			gvl.legCtrl[Mapping23[i]].ForwardKinetics(motorAngles:=OA_FJntRef[i].data , legIndex:=Mapping23[i] , tipPosition=>OA_FPosWrtHip[i].data );
			temp.data[0]:=hip_pos[Mapping23[i],0];temp.data[1]:=hip_pos[Mapping23[i],1];temp.data[2]:=hip_pos[Mapping23[i],2];
			leg_ref_pos[Mapping23[i]]:= VecAdd( MatMulVec(Rb_target1, VecAdd(temp,MatMulVec(Rleg[Mapping23[i]],OA_FPosWrtHip[i]))),body_ref_pos);	
		END_FOR		
	ELSE
		body_ref_pos:=OA_BodyPoseEnd;
		body_ref_ang:=OA_BodyAngEnd;
		leg_ref_pos:=OA_legPosEnterExtract;	
		tr  := (UDINT_TO_LREAL(gait_cycle - EnterOrientAdjustCount) / gvl.sampleRate-2*OA_LiftGroundTime-OA_AdjustTime-OA_AdjustExtractTime )/OA_AdjustExtendTime;
		fbGetPivot(tNow := tr, tTotal := 1.0, pivot => pvt);
		FOR i:=0 TO 1 DO
			FOR j:=0 TO 2 DO
				OA_MJntRef[i].data[j]:=(1-pvt)*OA_MJntExtract[i,j]+pvt*OA_MJntExtend[i,j];
			END_FOR		
			gvl.legCtrl[Mapping14[i]].ForwardKinetics(motorAngles:=OA_MJntRef[i].data , legIndex:=Mapping14[i] , tipPosition=>OA_MPosWrtHip[i].data );
			fbRotMat(yaw := body_ref_ang.data[2], pitch := body_ref_ang.data[1],roll := body_ref_ang.data[0], rm =>  Rb_target1 );
			temp.data[0]:=hip_pos[Mapping14[i],0];temp.data[1]:=hip_pos[Mapping14[i],1];temp.data[2]:=hip_pos[Mapping14[i],2];
			leg_ref_pos[Mapping14[i]]:= VecAdd( MatMulVec(Rb_target1, VecAdd(temp,MatMulVec(Rleg[Mapping14[i]],OA_MPosWrtHip[i]))),body_ref_pos);	

			gvl.legCtrl[Mapping23[i]].ForwardKinetics(motorAngles:=OA_FJntRef[i].data , legIndex:=Mapping23[i] , tipPosition=>OA_FPosWrtHip[i].data );
			temp.data[0]:=hip_pos[Mapping23[i],0];temp.data[1]:=hip_pos[Mapping23[i],1];temp.data[2]:=hip_pos[Mapping23[i],2];
			leg_ref_pos[Mapping23[i]]:= VecAdd( MatMulVec(Rb_target1, VecAdd(temp,MatMulVec(Rleg[Mapping23[i]],OA_FPosWrtHip[i]))),body_ref_pos);		
		END_FOR					
	END_IF
ELSE
	OrientAdjustFinished:=TRUE;
END_IF
END_METHOD

METHOD PUBLIC TrjPlanning_PushReleaseBall : BOOL
VAR_INPUT
END_VAR

VAR
	PushReleaseBall_FJntTarget:ARRAY[0..1,0..2] OF LREAL:=[-90*pi/180,155*pi/180,175*pi/180,
                                                     90*pi/180,155*pi/180,175*pi/180];//prepared position before gripping stone													 
													 
	i,j: INT;
	invalid: LREAL;
	Rb_target1: Mat3;
	temp: vec3;
	flag: INT;
	tr: LREAL;
END_VAR
//push and release method
IF PushReleaseBallFinished=FALSE AND gvl.curlingPushModel=0 THEN
	body_ref_pos:=body_ref_pos_enter;
	body_ref_ang:=body_ref_ang_enter;
	leg_ref_pos:=leg_ref_pos_enter;
	FOR i:=0 TO 1 DO
		IF gait_cycle-EnterPushReleaseBallCount<=PushTime*gvl.sampleRate THEN
			fbHermitInterpolation(t0:=EnterPushReleaseBallCount*delta_t , T:=PushTime , y0:=PushReleaseBall_FPosStartWrtHip[i].data[0] , 
			y1:=PushReleaseBall_FPosStartWrtHip[i].data[0]-PushDistance , v0:=0 , v1:=-PushVelocity , tNow:=(gait_cycle)* delta_t, 
			y=> PushReleaseBall_FPosWrtHip[i].data[0], v=>invalid );
		ELSIF gait_cycle-EnterPushReleaseBallCount<=(PushTime+PRConstVelTime)*gvl.sampleRate THEN
			fbHermitInterpolation(t0:=EnterPushReleaseBallCount*delta_t+PushTime , T:=PRConstVelTime , y0:=PushReleaseBall_FPosStartWrtHip[i].data[0]-PushDistance , 
			y1:=PushReleaseBall_FPosStartWrtHip[i].data[0]-PushDistance-PRConstVelDistance , v0:=-PushVelocity , v1:= -PushVelocity, tNow:=gait_cycle* delta_t, 
			y=> PushReleaseBall_FPosWrtHip[i].data[0], v=>invalid );			
		ELSIF gait_cycle-EnterPushReleaseBallCount<=(PushTime+PRConstVelTime+DecVelTime)*gvl.sampleRate THEN
			fbHermitInterpolation(t0:=EnterPushReleaseBallCount*delta_t+PushTime+PRConstVelTime , T:=DecVelTime , y0:=PushReleaseBall_FPosStartWrtHip[i].data[0]-PushDistance-PRConstVelDistance , 
			y1:=PushReleaseBall_FPosStartWrtHip[i].data[0]-PushDistance-PRConstVelDistance-DecVelDistance , v0:=-PushVelocity , v1:= 0, tNow:=gait_cycle* delta_t, 
			y=> PushReleaseBall_FPosWrtHip[i].data[0], v=>invalid );	
		ELSE
			 PushReleaseBall_FPosWrtHip[i].data[0]:=PushReleaseBall_FPosStartWrtHip[i].data[0]-PushDistance-PRConstVelDistance-DecVelDistance;	
			 PushReleaseBallFinished:=TRUE;	
			 EnterPushFinishCount:=gait_cycle;
			 
		END_IF
		PushReleaseBall_FPosWrtHip[i].data[1]:=PushReleaseBall_FPosStartWrtHip[i].data[1];
		PushReleaseBall_FPosWrtHip[i].data[2]:=PushReleaseBall_FPosStartWrtHip[i].data[2];
		
		fbRotMat(yaw := body_ref_ang_enter.data[2], pitch := body_ref_ang_enter.data[1],roll := body_ref_ang_enter.data[0], rm =>  Rb_target1 );
		temp.data[0]:=hip_pos[Mapping23[i],0];temp.data[1]:=hip_pos[Mapping23[i],1];temp.data[2]:=hip_pos[Mapping23[i],2];
		leg_ref_pos[Mapping23[i]]:= VecAdd( MatMulVec(Rb_target1, VecAdd(temp,MatMulVec(Rleg[Mapping23[i]],PushReleaseBall_FPosWrtHip[i]))),body_ref_pos);
	END_FOR
END_IF



//only release method
IF PushReleaseBallFinished=FALSE AND gvl.curlingPushModel=1 THEN
	IF gait_cycle - EnterPushReleaseBallCount<=ReleaseTime*gvl.sampleRate THEN
		body_ref_pos:=body_ref_pos_enter;
		body_ref_ang:=body_ref_ang_enter;
		leg_ref_pos:=leg_ref_pos_enter;
	
		tr  := UDINT_TO_LREAL(gait_cycle - EnterPushReleaseBallCount) / gvl.sampleRate / ReleaseTime;
		fbGetPivot(tNow := tr, tTotal := 1.0, pivot => pvt);
		FOR i:=0 TO 1 DO
			FOR j:=0 TO 2 DO
				PushReleaseBall_FJntRef[i].data[j]:=(1-pvt)*PushReleaseBall_FJntStart[i].data[j]+pvt*(PushReleaseBall_FJntTarget[i,j]);
			END_FOR
			gvl.legCtrl[Mapping23[i]].ForwardKinetics(motorAngles:=PushReleaseBall_FJntRef[i].data , legIndex:=Mapping23[i] , tipPosition=>PushReleaseBall_FPosWrtHip[i].data );
			fbRotMat(yaw := body_ref_ang_enter.data[2], pitch := body_ref_ang_enter.data[1],roll := body_ref_ang_enter.data[0], rm =>  Rb_target1 );
			temp.data[0]:=hip_pos[Mapping23[i],0];temp.data[1]:=hip_pos[Mapping23[i],1];temp.data[2]:=hip_pos[Mapping23[i],2];
			leg_ref_pos[Mapping23[i]]:= VecAdd( MatMulVec(Rb_target1, VecAdd(temp,MatMulVec(Rleg[Mapping23[i]],PushReleaseBall_FPosWrtHip[i]))),body_ref_pos);
		END_FOR
	ELSE	
		PushReleaseBallFinished:=TRUE;
		EnterPushFinishCount:=gait_cycle;
	END_IF	
END_IF

IF PushReleaseBallFinished=TRUE AND SpeedDownFinished=FALSE AND gait_cycle-EnterPushFinishCount>=LREAL_TO_UDINT(PushFinishDurationTime)*gvl.sampleRate  THEN
	RequireSpeedDown:=TRUE;
END_IF
END_METHOD

METHOD PUBLIC TrjPlanning_Recovery : BOOL
VAR_INPUT
END_VAR
VAR
	legExtractRefPosCurling: ARRAY[0..5, 0..2] OF LREAL:=[-0.35,-0.3+0.02,0,
														  0.1,-0.3+0.02,-0.1246,
														  -0.3+0.05,-0.3+0.02,-0.1246,
														  -0.3+0.05,-0.3+0.02,0.1246,
														  0.1,-0.3+0.02,0.1246,
														  -0.35,-0.3+0.02,0];//-0.15 for front leg
	jntExtractRefPosCurling: ARRAY[0..5, 0..2] OF LREAL:=[0,163.1808*pi/180,297.208*pi/180,
											  			  0,322.9120*pi/180,(205.1705-322.9120)*pi/180,
											              0,183.8227*pi/180,(269.8634-183.8227)*pi/180,
											              0,183.8227*pi/180,(269.8634-183.8227)*pi/180,
											              0,322.9120*pi/180,(205.1705-322.9120)*pi/180,
											              0,163.1808*pi/180,297.208*pi/180];
	legExtendRefPosCurling: ARRAY[0..5, 0..2] OF LREAL:=[-0.35,-0.4-0.07,0,
														  0.1,-0.4-0.07,-0.1246,
														  -0.3+0.05,-0.4-0.07,-0.1246,
														  -0.3+0.05,-0.4-0.07,0.1246,
														  0.1,-0.4-0.07,0.1246,
														  -0.35,-0.4-0.07,0];	//-0.15 for front leg													 
	jntExtendRefPosCurling: ARRAY[0..5, 0..2] OF LREAL:=[0,181.9845*pi/180,299.9603*pi/180,
											 			 0,302.7132*pi/180,(230.9946-302.7132)*pi/180,	
											             0,222.0252*pi/180,(254.0072-222.0252)*pi/180,
											             0,222.0252*pi/180,(254.0072-222.0252)*pi/180,
									                     0,302.7132*pi/180,(230.9946-302.7132)*pi/180,
											             0,181.9845*pi/180,299.9603*pi/180]	;

	(*legExtractRefPosCurling:    ARRAY[0..5, 0..2] OF LREAL:=[-0.35,-0.3+0.08,0,
														  0.1,-0.3209+0.08,-0.1246,
														  -0.3,-0.3209+0.08,-0.1246,
														  -0.3,-0.3209+0.08,0.1246,
														  0.1,-0.3209+0.08,0.1246,
														  -0.35,-0.3+0.08,0];															  
	jntExtractRefPosCurling: ARRAY[0..5, 0..2] OF LREAL:= [0,150.7997*pi/180,291.8958*pi/180,
											  			0,327.8142*pi/180,(196.8366-327.8142)*pi/180,
											  			0,172.5134*pi/180,(269.4767-172.5134)*pi/180,
											  			0,172.5134*pi/180,(269.4767-172.5134)*pi/180,
											  			0,327.8142*pi/180,(196.8366-327.8142)*pi/180,
											  			0,150.7997*pi/180,291.8958*pi/180];	
	legExtendRefPosCurling: ARRAY[0..5, 0..2] OF LREAL    :=[-0.35,-0.3209,0,
														  0.1,-0.3209,-0.1246,
														  -0.3,-0.3209,-0.1246,
														  -0.3,-0.3209,0.1246,
														  0.1,-0.3209,0.1246,
														  -0.35,-0.3209,0];														  													  
	jntExtendRefPosCurling: ARRAY[0..5, 0..2] OF LREAL:=	[0,163.1808*pi/180,297.208*pi/180,
											 				0,320.9331*pi/180,(208.0880-320.9331)*pi/180,	
											 				0,187.8384*pi/180,(269.4264-187.8384)*pi/180,
															0,187.8384*pi/180,(269.4264-187.8384)*pi/180,
									         				0,320.9331*pi/180,(208.0880-320.9331)*pi/180,
											 				0,163.1808*pi/180,297.208*pi/180];*)
													  
	i: INT;
	j: INT;
	tempLeg:ARRAY [0..2] OF LREAL;
	tempJnt:ARRAY [0..2] OF LREAL;
	tempRef:ARRAY [0..2] OF LREAL;
	tTotal: LREAL;
	tNow: LREAL;
	jntPosBegin : ARRAY[0..5, 0..2] OF LREAL;
	jntPosEnd   : ARRAY[0..5, 0..2] OF LREAL;
	Rb_target1: Mat3;
	temp: vec3;
	tipForceDesireGroupA:ARRAY[0..5,0..2] OF LREAL:=[0,-100,0,
													 0,0,0,
													 0,0,0,
													 0,0,0,
													 0,0,0,
													 0,0,0];
	tipForceDesireGroupB:ARRAY[0..5,0..2] OF LREAL:=[0,0,0,
													 0,0,0,
													 0,0,0,
													 0,0,0,
													 0,0,0,
													 0,-120,0];
	tr: LREAL;
END_VAR
IF (gait_cycle-EnterRecoveryCount)=1 THEN
	FOR i:=0 TO 5 DO
		tempLeg[0]:=legExtractRefPosCurling[i,0];tempLeg[1]:=legExtractRefPosCurling[i,1];tempLeg[2]:=legExtractRefPosCurling[i,2];
		tempRef[0]:=jntExtractRefPosCurling[i,0];tempRef[1]:=jntExtractRefPosCurling[i,1];tempRef[2]:=jntExtractRefPosCurling[i,2];
		GVL.legCtrl[i].InverseKinetics(tipPosition:=tempLeg , refPosLast:=tempRef , legIndex:=i , motorAngles=>tempJnt , isSingular=> );
		jntAngRetract[i,0]:=tempJnt[0];jntAngRetract[i,1]:=tempJnt[1];jntAngRetract[i,2]:=tempJnt[2];
		
		tempLeg[0]:=legExtendRefPosCurling[i,0];tempLeg[1]:=legExtendRefPosCurling[i,1];tempLeg[2]:=legExtendRefPosCurling[i,2];
		tempRef[0]:=jntExtendRefPosCurling[i,0];tempRef[1]:=jntExtendRefPosCurling[i,1];tempRef[2]:=jntExtendRefPosCurling[i,2];
		GVL.legCtrl[i].InverseKinetics(tipPosition:=tempLeg , refPosLast:=tempRef , legIndex:=i , motorAngles=>tempJnt , isSingular=> );
		jntAngExtend[i,0]:=tempJnt[0];jntAngExtend[i,1]:=tempJnt[1];jntAngExtend[i,2]:=tempJnt[2];			
		
	END_FOR
	tipForceDesire:=tipForceDesireZeros;

END_IF

IF RecoveryFinished=FALSE THEN
	body_ref_pos:=body_ref_pos_enter;
	body_ref_ang:=body_ref_ang_enter;
	leg_ref_pos:=leg_ref_pos_enter;
	
	IF (gait_cycle-EnterRecoveryCount)<=(tRetract + tWait + tExtend) * gvl.sampleRate THEN //leg 0-2-4 recovery
		
		//force compensator****************************
		IF (gait_cycle-EnterRecoveryCount)<=fceLoadTime*gvl.sampleRate THEN
			tr  := UDINT_TO_LREAL(gait_cycle-EnterRecoveryCount) / gvl.sampleRate /fceLoadTime;
			fbGetPivot(tNow := tr, tTotal := 1.0, pivot => pvt);
			FOR i:=0 TO 5 DO
				FOR j:=0 TO 2 DO
					tipForceDesire[i,j]:=(1-pvt)*tipForceDesireZeros[i,j]+pvt*tipForceDesireGroupB[i,j];//group B add load
				END_FOR
			END_FOR
		ELSIF  (gait_cycle-EnterRecoveryCount)>LREAL_TO_UDINT((tRetract + tWait + tExtend-fceLoadTime)*gvl.sampleRate) AND  (gait_cycle-EnterRecoveryCount)<=LREAL_TO_UDINT((tRetract + tWait + tExtend) * gvl.sampleRate) THEN
			tr  := (UDINT_TO_LREAL (gait_cycle-EnterRecoveryCount) / gvl.sampleRate-(tRetract + tWait + tExtend-fceLoadTime) )/fceLoadTime;
			fbGetPivot(tNow := tr, tTotal := 1.0, pivot => pvt);
			FOR i:=0 TO 5 BY 2DO
				FOR j:=0 TO 2 DO
					//tipForceDesire[i,j]:=(1-pvt)*tipForceDesireZeros[i,j]+pvt*tipForceDesireGroupA[i,j];//group A add load
					tipForceDesire[i+1,j]:=(1-pvt)*tipForceDesireGroupB[i+1,j]+pvt*tipForceDesireZeros[i+1,j];//group B reduce load
				END_FOR
			END_FOR
		ELSE
		tipForceDesire:=tipForceDesireGroupB;
		END_IF
		//***********************************************
	
		IF gait_cycle-EnterRecoveryCount < tRetract * gvl.sampleRate THEN
			tTotal := tRetract;
			tNow   := UDINT_TO_LREAL(gait_cycle-EnterRecoveryCount) * 1.0 / DINT_TO_LREAL(gvl.sampleRate);
			jntPosBegin := RcJointPosStart;
			FOR i:=0 TO 5 BY 2 DO
				FOR j:=0 TO 2 DO
					jntPosEnd[i,j]:=jntAngRetract[i,j];
					jntPosEnd[i+1,j]:=RcJointPosStart[i+1,j];
				END_FOR
			END_FOR
		ELSIF gait_cycle-EnterRecoveryCount  < (tRetract + tWait) * gvl.sampleRate THEN
			tTotal := tWait;
			tNow   := UDINT_TO_LREAL(gait_cycle-EnterRecoveryCount) * 1.0 / DINT_TO_LREAL(gvl.sampleRate) - tRetract;
			FOR i:=0 TO 5 BY 2 DO
				FOR j:=0 TO 2 DO
					jntPosBegin[i,j]:=jntAngRetract[i,j];
					jntPosBegin[i+1,j]:=RcJointPosStart[i+1,j];
					jntPosEnd[i,j]:=jntAngRetract[i,j];
					jntPosEnd[i+1,j]:=RcJointPosStart[i+1,j];
				END_FOR
			END_FOR
		ELSE 
			tTotal := tExtend;
			tNow   := UDINT_TO_LREAL(gait_cycle-EnterRecoveryCount) * 1.0 / DINT_TO_LREAL(gvl.sampleRate) - tRetract - tWait;
			FOR i:=0 TO 5 BY 2 DO
				FOR j:=0 TO 2 DO
					jntPosBegin[i,j]:=jntAngRetract[i,j];
					jntPosBegin[i+1,j]:=RcJointPosStart[i+1,j];
					jntPosEnd[i,j]:=jntAngExtend[i,j];
					jntPosEnd[i+1,j]:=RcJointPosStart[i+1,j];
				END_FOR
			END_FOR	
		END_IF	
	ELSIF (gait_cycle-EnterRecoveryCount)<=2*(tRetract + tWait + tExtend) * gvl.sampleRate  THEN //leg 1-3-5 recovery

		//force compensator*******************
		IF (gait_cycle-EnterRecoveryCount)>LREAL_TO_UDINT((tRetract + tWait + tExtend)*gvl.sampleRate) AND (gait_cycle-EnterRecoveryCount)<=LREAL_TO_UDINT((tRetract + tWait + tExtend+fceLoadTime)* gvl.sampleRate) THEN
			tr  := (UDINT_TO_LREAL(gait_cycle-EnterRecoveryCount) / gvl.sampleRate-(tRetract + tWait + tExtend) )/fceLoadTime;
			fbGetPivot(tNow := tr, tTotal := 1.0, pivot => pvt);
			FOR i:=0 TO 5 BY 2 DO
				FOR j:=0 TO 2 DO
					tipForceDesire[i,j]:=(1-pvt)*tipForceDesireZeros[i,j]+pvt*tipForceDesireGroupA[i,j];//group A add load
					tipForceDesire[i+1,j]:=tipForceDesireZeros[i+1,j];//group B zeros load
				END_FOR
			END_FOR		
		ELSIF (gait_cycle-EnterRecoveryCount)>LREAL_TO_UDINT((2*(tRetract + tWait + tExtend)-fceLoadTime)*gvl.sampleRate) AND (gait_cycle-EnterRecoveryCount)<=LREAL_TO_UDINT(2*(tRetract + tWait + tExtend) * gvl.sampleRate) THEN
			tr  := (UDINT_TO_LREAL(gait_cycle-EnterRecoveryCount) / gvl.sampleRate-(2*(tRetract + tWait + tExtend)-fceLoadTime) )/fceLoadTime;
			fbGetPivot(tNow := tr, tTotal := 1.0, pivot => pvt);
			FOR i:=0 TO 5 BY 2DO
				FOR j:=0 TO 2 DO
					tipForceDesire[i,j]:=(1-pvt)*tipForceDesireGroupA[i,j]+pvt*tipForceDesireZeros[i,j];//group A reduce load
					tipForceDesire[i+1,j]:=tipForceDesireZeros[i+1,j];//group B zeros load
				END_FOR
			END_FOR	
		ELSE	
			tipForceDesire:=tipForceDesireGroupA;
		END_IF	
		//******************************************	

		
		IF gait_cycle-EnterRecoveryCount<=(2*tRetract + tWait + tExtend) * gvl.sampleRate THEN
			tTotal := tRetract;
			tNow   := UDINT_TO_LREAL(gait_cycle-EnterRecoveryCount) * 1.0 / DINT_TO_LREAL(gvl.sampleRate)-(tRetract + tWait + tExtend);
			FOR i:=0 TO 5 BY 2 DO
				FOR j:=0 TO 2 DO
					jntPosBegin[i,j]:=jntAngExtend[i,j];
					jntPosBegin[i+1,j]:=RcJointPosStart[i+1,j];
					jntPosEnd[i,j]:=jntAngExtend[i,j];
					jntPosEnd[i+1,j]:=jntAngRetract[i+1,j];
				END_FOR
			END_FOR			
		ELSIF gait_cycle-EnterRecoveryCount<=(2*tRetract + 2*tWait + tExtend) * gvl.sampleRate THEN
			tTotal := tWait;
			tNow   := UDINT_TO_LREAL(gait_cycle-EnterRecoveryCount) * 1.0 / DINT_TO_LREAL(gvl.sampleRate) - (2*tRetract + tWait + tExtend);
			FOR i:=0 TO 5 BY 2 DO
				FOR j:=0 TO 2 DO
					jntPosBegin[i,j]:=jntAngExtend[i,j];
					jntPosBegin[i+1,j]:=jntAngRetract[i+1,j];
					jntPosEnd[i,j]:=jntAngExtend[i,j];
					jntPosEnd[i+1,j]:=jntAngRetract[i+1,j];
				END_FOR
			END_FOR			
		ELSE
			tTotal := tExtend;
			tNow   := UDINT_TO_LREAL(gait_cycle-EnterRecoveryCount) * 1.0 / DINT_TO_LREAL(gvl.sampleRate) - (2*tRetract + 2*tWait + tExtend);
			FOR i:=0 TO 5 BY 2 DO
				FOR j:=0 TO 2 DO
					jntPosBegin[i,j]:=jntAngExtend[i,j];
					jntPosBegin[i+1,j]:=jntAngRetract[i+1,j];
					jntPosEnd[i,j]:=jntAngExtend[i,j];
					jntPosEnd[i+1,j]:=jntAngExtend[i+1,j];
				END_FOR
			END_FOR			
		END_IF
	ELSE
		tTotal := 100;
		tNow   := UDINT_TO_LREAL(gait_cycle-EnterRecoveryCount) * 1.0 / DINT_TO_LREAL(gvl.sampleRate) - 2*tRetract - 2*tWait - 2*tExtend;
		jntPosBegin :=jntAngExtend;
		jntPosEnd :=jntAngExtend;
		RecoveryFinished:=TRUE;
		tipForceDesire:=tipForceDesireZeros;
		RequireReduceHeightB:=TRUE;
	END_IF
	getPivot(tNow := tNow, tTotal := tTotal, pivot => pivot, pivotDot => pivotDot);
	FOR i := 0 TO 5 DO
		FOR j := 0 TO 2 DO
			RcJointPosRef[i, j] := (1.0 - pivot) * jntPosBegin[i, j] + pivot * jntPosEnd[i, j];
		END_FOR
		tempJnt[0]:=RcJointPosRef[i,0];tempJnt[1]:=RcJointPosRef[i,1];tempJnt[2]:=RcJointPosRef[i,2];
		gvl.legCtrl[i].ForwardKinetics(motorAngles:=tempJnt , legIndex:=i , tipPosition=>Rc_PosWrtHip[i].data );
		fbRotMat(yaw := body_ref_ang_enter.data[2], pitch := body_ref_ang_enter.data[1],roll := body_ref_ang_enter.data[0], rm =>  Rb_target1 );
		temp.data[0]:=hip_pos[i,0];temp.data[1]:=hip_pos[i,1];temp.data[2]:=hip_pos[i,2];
		leg_ref_pos[i]:= VecAdd( MatMulVec(Rb_target1, VecAdd(temp,MatMulVec(Rleg[i],Rc_PosWrtHip[i]))),body_ref_pos);		
	END_FOR

END_IF
END_METHOD

METHOD PUBLIC TrjPlanning_ReduceHeight : BOOL
VAR_INPUT
	
END_VAR
VAR
	
	tr: LREAL;
	i: INT;
	Rb_target1: Mat3;
	temp: vec3;
END_VAR
IF ReduceHeightFinished=FALSE AND (gait_cycle-EnterReduceHeightCount)<=ReduceHeightTime*gvl.sampleRate THEN
	body_ref_ang:=body_ref_ang_enter;
	leg_ref_pos:=leg_ref_pos_enter;
	tr  := UDINT_TO_LREAL(gait_cycle - EnterReduceHeightCount) / gvl.sampleRate / ReduceHeightTime;
	fbGetPivot(tNow := tr, tTotal := 1.0, pivot => pvt);
	FOR i:=0 TO 2 DO
		body_ref_pos.data[i]:=(1-pvt)*body_ref_pos_enter.data[i]+pvt*body_target_pos.data[i];
	END_FOR
	FOR i:=0 TO 1 DO
		gvl.legCtrl[Mapping23[i]].ForwardKinetics(motorAngles:=ReduceHeight_FJntRef[i].data , legIndex:=Mapping23[i] , tipPosition=>ReduceHeight_FPosWrtHip[i].data );
		fbRotMat(yaw := body_ref_ang_enter.data[2], pitch := body_ref_ang_enter.data[1],roll := body_ref_ang_enter.data[0], rm =>  Rb_target1 );
		temp.data[0]:=hip_pos[Mapping23[i],0];temp.data[1]:=hip_pos[Mapping23[i],1];temp.data[2]:=hip_pos[Mapping23[i],2];
		leg_ref_pos[Mapping23[i]]:= VecAdd( MatMulVec(Rb_target1, VecAdd(temp,MatMulVec(Rleg[Mapping23[i]],ReduceHeight_FPosWrtHip[i]))),body_ref_pos);
	END_FOR
ELSE
	ReduceHeightFinished:=TRUE;
END_IF
END_METHOD

METHOD PUBLIC TrjPlanning_ReduceHeightB : BOOL
VAR_INPUT
END_VAR
VAR
	tr: LREAL;
	i: INT;
	Rb_target1: Mat3;
	temp: vec3;
END_VAR
IF ReduceHeightBFinished=FALSE AND (gait_cycle-EnterReduceHeightBCount)<=RHB_time*gvl.sampleRate THEN
	body_ref_ang:=body_ref_ang_enter;
	leg_ref_pos:=leg_ref_pos_enter;
	tr  := UDINT_TO_LREAL(gait_cycle - EnterReduceHeightBCount) / gvl.sampleRate / RHB_time;
	fbGetPivot(tNow := tr, tTotal := 1.0, pivot => pvt);
	FOR i:=0 TO 2 DO
		body_ref_pos.data[i]:=(1-pvt)*body_ref_pos_enter.data[i]+pvt*RHB_body_target_pos.data[i];
	END_FOR
ELSE
	ReduceHeightBFinished:=TRUE;
END_IF
END_METHOD

METHOD PUBLIC TrjPlanning_SearchPedal : BOOL
VAR_INPUT
END_VAR
VAR
	tr: LREAL;
	i: INT;
	j: INT;
	Rb_target1: Mat3;
	temp: vec3;
	
	tipForceDesireLegA:	 ARRAY[0..5,0..2] OF LREAL:=[0,-100,0,
													 0,0,0,
													 0,0,0,
													 0,0,0,
													 0,0,0,
													 0,0,0];
	tipForceDesireLegF:	 ARRAY[0..5,0..2] OF LREAL:=[0,0,0,
													 0,0,0,
													 0,0,0,
													 0,0,0,
													 0,0,0,
													 0,-120,0];				
END_VAR
IF SearchPedalFinished=FALSE THEN
	IF SP_RBLegSearching=TRUE THEN
		SP_LBLegSearching:=FALSE;
		body_ref_pos:=body_ref_pos_enter;
		body_ref_ang:=body_ref_ang_enter;
		leg_ref_pos:=leg_ref_pos_enter;	
		IF (gait_cycle-SP_EnterSubSearchCount[0])<=SP_LiftLegTime*gvl.sampleRate THEN
			tr  := UDINT_TO_LREAL(gait_cycle - SP_EnterSubSearchCount[0]) / gvl.sampleRate / SP_LiftLegTime;
			fbGetPivot(tNow := tr, tTotal := 1.0, pivot => pvt);	
			SP_BPosRefWrtHip[0].data[0]:=SP_BPosStartWrtHip[0].data[0];
			SP_BPosRefWrtHip[0].data[1]:=(1-pvt)*SP_BPosStartWrtHip[0].data[1]+pvt*(SP_BPosStartWrtHip[0].data[1]+SP_LiftDistance);
			SP_BPosRefWrtHip[0].data[2]:=SP_BPosStartWrtHip[0].data[2];
			fbRotMat(yaw := body_ref_ang_enter.data[2], pitch := body_ref_ang_enter.data[1],roll := body_ref_ang_enter.data[0], rm =>  Rb_target1 );
			temp.data[0]:=hip_pos[0,0];temp.data[1]:=hip_pos[0,1];temp.data[2]:=hip_pos[0,2];
			leg_ref_pos[0]:= VecAdd( MatMulVec(Rb_target1, VecAdd(temp,MatMulVec(Rleg[0],SP_BPosRefWrtHip[0]))),body_ref_pos);	
			
			//force compensator
			tipForceTarget:=tipForceDesireLegF;
			IF (gait_cycle-SP_EnterSubSearchCount[0])<=LREAL_TO_UDINT(fceLoadTime*gvl.sampleRate) THEN
				tr  := (UDINT_TO_LREAL(gait_cycle-SP_EnterSubSearchCount[0]) / gvl.sampleRate)/ fceLoadTime;
				fbGetPivot(tNow := tr, tTotal := 1.0, pivot => pvt);
				FOR i:=0 TO 5 DO
					FOR j:=0 TO 2 DO
						tipForceDesire[i,j]:=(1-pvt)*tipForceDesireZeros[i,j]+pvt*tipForceTarget[i,j];
					END_FOR
				END_FOR
			END_IF
			
		ELSIF (gait_cycle-SP_EnterSubSearchCount[0])<=(SP_LiftLegTime+SP_SearchTime)*gvl.sampleRate AND  SP_BLegSearchFinished[0]=FALSE THEN
			tr  := (UDINT_TO_LREAL(gait_cycle - SP_EnterSubSearchCount[0]) / gvl.sampleRate -SP_LiftLegTime)/ SP_SearchTime;
			fbGetPivot(tNow := tr, tTotal := 1.0, pivot => pvt);	
			SP_BPosRefWrtHip[0].data[0]:=(1-pvt)*SP_BPosStartWrtHip[0].data[0]+pvt*(SP_BPosStartWrtHip[0].data[0]-SP_SearchDistance);		
			SP_BPosRefWrtHip[0].data[1]:=SP_BPosStartWrtHip[0].data[1]+SP_LiftDistance;
			SP_BPosRefWrtHip[0].data[2]:=SP_BPosStartWrtHip[0].data[2];
			IF isPedal(0)=TRUE AND  SP_BLegSearchFinished[0]=FALSE THEN
				SP_BLegSearchFinished[0]:=TRUE;
				SP_EnterSubSearchDecreaseCount[0]:=gait_cycle;
				FOR j:=0 TO 2 DO
					SP_BPosLockWrtHip[0].data[j]:=SP_BPosRefWrtHip[0].data[j];
				END_FOR			
			END_IF
			IF (gait_cycle-SP_EnterSubSearchCount[0])=LREAL_TO_UDINT((SP_LiftLegTime+SP_SearchTime)*gvl.sampleRate) AND SP_BLegSearchFinished[0]=FALSE THEN
				SP_BLegSearchFinished[0]:=TRUE;
				SP_EnterSubSearchDecreaseCount[0]:=gait_cycle;
				FOR j:=0 TO 2 DO
					SP_BPosLockWrtHip[0].data[j]:=SP_BPosRefWrtHip[0].data[j];
				END_FOR	
			END_IF

			fbRotMat(yaw := body_ref_ang_enter.data[2], pitch := body_ref_ang_enter.data[1],roll := body_ref_ang_enter.data[0], rm =>  Rb_target1 );
			temp.data[0]:=hip_pos[0,0];temp.data[1]:=hip_pos[0,1];temp.data[2]:=hip_pos[0,2];
			leg_ref_pos[0]:= VecAdd( MatMulVec(Rb_target1, VecAdd(temp,MatMulVec(Rleg[0],SP_BPosRefWrtHip[0]))),body_ref_pos);	
			
		ELSIF  SP_BLegSearchFinished[0]=TRUE AND (gait_cycle-SP_EnterSubSearchDecreaseCount[0])<=SP_LiftLegTime*gvl.sampleRate THEN
			tr  := UDINT_TO_LREAL(gait_cycle - SP_EnterSubSearchDecreaseCount[0]) / gvl.sampleRate / SP_LiftLegTime;
			fbGetPivot(tNow := tr, tTotal := 1.0, pivot => pvt);
			SP_BPosRefWrtHip[0].data[0]:=SP_BPosLockWrtHip[0].data[0];	
			SP_BPosRefWrtHip[0].data[1]:=(1-pvt)*SP_BPosLockWrtHip[0].data[1]+pvt*(SP_BPosLockWrtHip[0].data[1]-SP_LiftDistance);
			SP_BPosRefWrtHip[0].data[2]:=SP_BPosLockWrtHip[0].data[2];	
			
			fbRotMat(yaw := body_ref_ang_enter.data[2], pitch := body_ref_ang_enter.data[1],roll := body_ref_ang_enter.data[0], rm =>  Rb_target1 );
			temp.data[0]:=hip_pos[0,0];temp.data[1]:=hip_pos[0,1];temp.data[2]:=hip_pos[0,2];
			leg_ref_pos[0]:= VecAdd( MatMulVec(Rb_target1, VecAdd(temp,MatMulVec(Rleg[0],SP_BPosRefWrtHip[0]))),body_ref_pos);	
			IF (gait_cycle-SP_EnterSubSearchDecreaseCount[0])=LREAL_TO_UDINT( SP_LiftLegTime*gvl.sampleRate) THEN
				body_ref_pos_enter:=body_ref_pos;
				body_ref_ang_enter:=body_ref_ang;
				leg_ref_pos_enter:=leg_ref_pos;	
			END_IF	
			
			//force compensator
			tipForceTarget:=tipForceDesireLegF;
			IF (gait_cycle-SP_EnterSubSearchDecreaseCount[0])>LREAL_TO_UDINT((SP_LiftLegTime-fceLoadTime)*gvl.sampleRate)THEN
				tr  := (UDINT_TO_LREAL(gait_cycle-SP_EnterSubSearchDecreaseCount[0]) / gvl.sampleRate-(SP_LiftLegTime-fceLoadTime) )/ fceLoadTime;
				fbGetPivot(tNow := tr, tTotal := 1.0, pivot => pvt);
				FOR i:=0 TO 5 DO
					FOR j:=0 TO 2 DO
						tipForceDesire[i,j]:=(1-pvt)*tipForceTarget[i,j]+pvt*tipForceDesireZeros[i,j];
					END_FOR
				END_FOR
			END_IF
	
		ELSE
			SP_RBLegSearching:=FALSE;
			SP_LBLegSearching:=TRUE;
			SP_EnterSubSearchCount[1]:=gait_cycle;			
		END_IF
	END_IF
	
	IF SP_LBLegSearching=TRUE THEN
		SP_RBLegSearching:=FALSE;
		body_ref_pos:=body_ref_pos_enter;
		body_ref_ang:=body_ref_ang_enter;
		leg_ref_pos:=leg_ref_pos_enter;	
		IF (gait_cycle-SP_EnterSubSearchCount[1])<=SP_LiftLegTime*gvl.sampleRate THEN
			tr  := UDINT_TO_LREAL(gait_cycle - SP_EnterSubSearchCount[1]) / gvl.sampleRate / SP_LiftLegTime;
			fbGetPivot(tNow := tr, tTotal := 1.0, pivot => pvt);	
			SP_BPosRefWrtHip[1].data[0]:=SP_BPosStartWrtHip[1].data[0];
			SP_BPosRefWrtHip[1].data[1]:=(1-pvt)*SP_BPosStartWrtHip[1].data[1]+pvt*(SP_BPosStartWrtHip[1].data[1]+SP_LiftDistance);
			SP_BPosRefWrtHip[1].data[2]:=SP_BPosStartWrtHip[1].data[2];
			fbRotMat(yaw := body_ref_ang_enter.data[2], pitch := body_ref_ang_enter.data[1],roll := body_ref_ang_enter.data[0], rm =>  Rb_target1 );
			temp.data[0]:=hip_pos[5,0];temp.data[1]:=hip_pos[5,1];temp.data[2]:=hip_pos[5,2];
			leg_ref_pos[5]:= VecAdd( MatMulVec(Rb_target1, VecAdd(temp,MatMulVec(Rleg[5],SP_BPosRefWrtHip[1]))),body_ref_pos);	
			
			//force compensator
			tipForceTarget:=tipForceDesireLegA;
			IF (gait_cycle-SP_EnterSubSearchCount[1])<=LREAL_TO_UDINT(fceLoadTime*gvl.sampleRate) THEN
				tr  := (UDINT_TO_LREAL(gait_cycle-SP_EnterSubSearchCount[1]) / gvl.sampleRate)/ fceLoadTime;
				fbGetPivot(tNow := tr, tTotal := 1.0, pivot => pvt);
				FOR i:=0 TO 5 DO
					FOR j:=0 TO 2 DO
						tipForceDesire[i,j]:=(1-pvt)*tipForceDesireZeros[i,j]+pvt*tipForceTarget[i,j];
					END_FOR
				END_FOR
			END_IF
			
		ELSIF (gait_cycle-SP_EnterSubSearchCount[1])<=(SP_LiftLegTime+SP_SearchTime)*gvl.sampleRate AND  SP_BLegSearchFinished[1]=FALSE THEN
			tr  := (UDINT_TO_LREAL(gait_cycle - SP_EnterSubSearchCount[1]) / gvl.sampleRate -SP_LiftLegTime)/ SP_SearchTime;
			fbGetPivot(tNow := tr, tTotal := 1.0, pivot => pvt);	
			SP_BPosRefWrtHip[1].data[0]:=(1-pvt)*SP_BPosStartWrtHip[1].data[0]+pvt*(SP_BPosStartWrtHip[1].data[0]-SP_SearchDistance);		
			SP_BPosRefWrtHip[1].data[1]:=SP_BPosStartWrtHip[1].data[1]+SP_LiftDistance;
			SP_BPosRefWrtHip[1].data[2]:=SP_BPosStartWrtHip[1].data[2];
			IF isPedal(5)=TRUE AND  SP_BLegSearchFinished[1]=FALSE THEN
				SP_BLegSearchFinished[1]:=TRUE;
				SP_EnterSubSearchDecreaseCount[1]:=gait_cycle;
				FOR j:=0 TO 2 DO
					SP_BPosLockWrtHip[1].data[j]:=SP_BPosRefWrtHip[1].data[j];
				END_FOR			
			END_IF
			IF (gait_cycle-SP_EnterSubSearchCount[1])=LREAL_TO_UDINT((SP_LiftLegTime+SP_SearchTime)*gvl.sampleRate) AND SP_BLegSearchFinished[1]=FALSE THEN
				SP_BLegSearchFinished[1]:=TRUE;
				SP_EnterSubSearchDecreaseCount[1]:=gait_cycle;
				FOR j:=0 TO 2 DO
					SP_BPosLockWrtHip[1].data[j]:=SP_BPosRefWrtHip[1].data[j];
				END_FOR	
			END_IF

			fbRotMat(yaw := body_ref_ang_enter.data[2], pitch := body_ref_ang_enter.data[1],roll := body_ref_ang_enter.data[0], rm =>  Rb_target1 );
			temp.data[0]:=hip_pos[5,0];temp.data[1]:=hip_pos[5,1];temp.data[2]:=hip_pos[5,2];
			leg_ref_pos[5]:= VecAdd( MatMulVec(Rb_target1, VecAdd(temp,MatMulVec(Rleg[5],SP_BPosRefWrtHip[1]))),body_ref_pos);	
			
		ELSIF  SP_BLegSearchFinished[1]=TRUE AND (gait_cycle-SP_EnterSubSearchDecreaseCount[1])<=SP_LiftLegTime*gvl.sampleRate THEN
			tr  := UDINT_TO_LREAL(gait_cycle - SP_EnterSubSearchDecreaseCount[1]) / gvl.sampleRate / SP_LiftLegTime;
			fbGetPivot(tNow := tr, tTotal := 1.0, pivot => pvt);
			SP_BPosRefWrtHip[1].data[0]:=SP_BPosLockWrtHip[1].data[0];	
			SP_BPosRefWrtHip[1].data[1]:=(1-pvt)*SP_BPosLockWrtHip[1].data[1]+pvt*(SP_BPosLockWrtHip[1].data[1]-SP_LiftDistance);
			SP_BPosRefWrtHip[1].data[2]:=SP_BPosLockWrtHip[1].data[2];	
			
			fbRotMat(yaw := body_ref_ang_enter.data[2], pitch := body_ref_ang_enter.data[1],roll := body_ref_ang_enter.data[0], rm =>  Rb_target1 );
			temp.data[0]:=hip_pos[5,0];temp.data[1]:=hip_pos[5,1];temp.data[2]:=hip_pos[5,2];
			leg_ref_pos[5]:= VecAdd( MatMulVec(Rb_target1, VecAdd(temp,MatMulVec(Rleg[5],SP_BPosRefWrtHip[1]))),body_ref_pos);	
			IF (gait_cycle-SP_EnterSubSearchDecreaseCount[1])=LREAL_TO_UDINT( SP_LiftLegTime*gvl.sampleRate) THEN
				body_ref_pos_enter:=body_ref_pos;
				body_ref_ang_enter:=body_ref_ang;
				leg_ref_pos_enter:=leg_ref_pos;	
			END_IF	
			
			//force compensator
			tipForceTarget:=tipForceDesireLegA;
			IF (gait_cycle-SP_EnterSubSearchDecreaseCount[1])>LREAL_TO_UDINT((SP_LiftLegTime-fceLoadTime)*gvl.sampleRate)THEN
				tr  := (UDINT_TO_LREAL(gait_cycle-SP_EnterSubSearchDecreaseCount[1]) / gvl.sampleRate-(SP_LiftLegTime-fceLoadTime) )/ fceLoadTime;
				fbGetPivot(tNow := tr, tTotal := 1.0, pivot => pvt);
				FOR i:=0 TO 5 DO
					FOR j:=0 TO 2 DO
						tipForceDesire[i,j]:=(1-pvt)*tipForceTarget[i,j]+pvt*tipForceDesireZeros[i,j];
					END_FOR
				END_FOR
			END_IF			
			
		ELSE
			SP_RBLegSearching:=FALSE;
			SP_LBLegSearching:=FALSE;	
			SearchPedalFinished:=TRUE;	
			tipForceDesire:=tipForceDesireZeros;
		END_IF
	END_IF	
END_IF
END_METHOD

METHOD PUBLIC TrjPlanning_Slide : BOOL
VAR_INPUT
END_VAR
IF SlideFinished=FALSE THEN
	body_ref_pos:=body_ref_pos_enter;
	body_ref_ang:=body_ref_ang_enter;
	leg_ref_pos:=leg_ref_pos_enter;

END_IF

//***********tuning***************************
IF SlideFinished=FALSE AND (gait_cycle-EnterSlideCount)>=LREAL_TO_UDINT(slideTime*gvl.sampleRate) THEN
	RequirePushReleaseBall:=TRUE;
END_IF

//*************end-tuning********************



IF SlideFinished=FALSE AND RequirePushReleaseBall=TRUE THEN
	SlideFinished:=TRUE;
END_IF
END_METHOD

METHOD PUBLIC TrjPlanning_SpeedDown : BOOL
VAR_INPUT
END_VAR

VAR
	tr: LREAL;
	i: INT;
	SpeedDown_MPosTarget:ARRAY[0..1,0..2] OF LREAL:=[-0.0141,-0.1797,-0.1246,
                                                        -0.0141,-0.1797,0.1246];
	SpeedDown_MJntTargetRef:ARRAY[0..1,0..2] OF LREAL:=[0,331.45*pi/180,-144*pi/180,
                                                     0,331.45*pi/180,-144*pi/180];
	j: INT;
	Rb_target1: Mat3;
	temp: vec3;
	tempLeg:ARRAY [0..2] OF LREAL;
	tempJnt:ARRAY [0..2] OF LREAL;
	tempRef:ARRAY [0..2] OF LREAL;
END_VAR
IF (gait_cycle-EnterSpeedDownCount)=1 THEN
	FOR i:=0 TO 1 DO
		tempLeg[0]:=SpeedDown_MPosTarget[i,0];tempLeg[1]:=SpeedDown_MPosTarget[i,1];tempLeg[2]:=SpeedDown_MPosTarget[i,2];
		tempRef[0]:=SpeedDown_MJntTargetRef[i,0];tempRef[1]:=SpeedDown_MJntTargetRef[i,1];tempRef[2]:=SpeedDown_MJntTargetRef[i,2];
		GVL.legCtrl[Mapping14[i]].InverseKinetics(tipPosition:=tempLeg , refPosLast:=tempRef , legIndex:=Mapping14[i] , motorAngles=>tempJnt , isSingular=> );
		SpeedDown_MJntTarget[i,0]:=tempJnt[0];SpeedDown_MJntTarget[i,1]:=tempJnt[1];SpeedDown_MJntTarget[i,2]:=tempJnt[2];		
	END_FOR
END_IF

IF SpeedDownFinished=FALSE THEN
	IF gait_cycle-EnterSpeedDownCount<=SpeedDownTime*gvl.sampleRate THEN
		body_ref_pos:=body_ref_pos_enter;
		body_ref_ang:=body_ref_ang_enter;
		leg_ref_pos:=leg_ref_pos_enter;
		tr  := UDINT_TO_LREAL(gait_cycle - EnterSpeedDownCount) / gvl.sampleRate / SpeedDownTime;
		fbGetPivot(tNow := tr, tTotal := 1.0, pivot => pvt);
		FOR i:=0 TO 1 DO
			FOR j:=0 TO 2 DO
				SpeedDown_MJntRef[i].data[j]:=(1-pvt)*SpeedDown_MJntStart[i].data[j]+pvt*SpeedDown_MJntTarget[i,j];
			END_FOR
			gvl.legCtrl[Mapping14[i]].ForwardKinetics(motorAngles:=SpeedDown_MJntRef[i].data , legIndex:=Mapping14[i] , tipPosition=>SpeedDown_MPosWrtHip[i].data );
			fbRotMat(yaw := body_ref_ang_enter.data[2], pitch := body_ref_ang_enter.data[1],roll := body_ref_ang_enter.data[0], rm =>  Rb_target1 );
			temp.data[0]:=hip_pos[Mapping14[i],0];temp.data[1]:=hip_pos[Mapping14[i],1];temp.data[2]:=hip_pos[Mapping14[i],2];
			leg_ref_pos[Mapping14[i]]:= VecAdd( MatMulVec(Rb_target1, VecAdd(temp,MatMulVec(Rleg[Mapping14[i]],SpeedDown_MPosWrtHip[i]))),body_ref_pos);
			
			leg_ref_pos[Mapping05[i]].data[2]:=(1-pvt)*leg_ref_pos_enter[Mapping05[i]].data[2]+pvt*(leg_ref_pos_enter[Mapping05[i]].data[2]-Distance_y_DS-0.005);
		END_FOR
	ELSE
		SpeedDownFinished:=TRUE;
		
	END_IF
	
	IF gait_cycle-EnterSpeedDownCount=1 THEN
		GVL.jogVelocity[18]:=0;
		GVL.jogVelocity[19]:=0;
		gvl.jogStopButton[18]:=TRUE;
		gvl.jogStopButton[19]:=TRUE;
		gvl.motorDrive[j].SetTrgVel(0);
	END_IF
END_IF
END_METHOD

METHOD PUBLIC TrjPlanning_SpeedUp : BOOL
VAR_INPUT
END_VAR

VAR
	invalid: LREAL;
	Rb_target1: Mat3;
	i: INT;
	tr: LREAL;
	temp: VEC3;
	
	
	tipForceDesireLegAF:	 ARRAY[0..5,0..2] OF LREAL:=[0,-5,0,
													 0,0,0,
													 0,0,0,
													 0,0,0,
													 0,0,0,
													 0,-5,0];
	j: INT;
END_VAR
IF SpeedUpSubState=SpeedUpAS AND (gait_cycle-EnterSpeedUpASCount)=LREAL_TO_UDINT(Time_AS*gvl.sampleRate) THEN
	SpeedUpSubState:=SpeedUpCS;
	EnterSpeedUpCSCount:=gait_cycle;
	body_ref_pos_enter :=body_ref_pos;
	body_ref_ang_enter:=body_ref_ang;
	leg_ref_pos_enter := leg_ref_pos;
	
ELSIF SpeedUpSubState=SpeedUpCS AND gait_cycle-EnterSpeedUpCSCount=LREAL_TO_UDINT(Time_CS*gvl.sampleRate) THEN
	SpeedUpSubState:=SpeedUpDS;
	EnterSpeedUpDSCount:=gait_cycle;
	body_ref_pos_enter :=body_ref_pos;
	body_ref_ang_enter:=body_ref_ang;
	leg_ref_pos_enter := leg_ref_pos;
ELSIF SpeedUpSubState=SpeedUpDS AND gait_cycle-EnterSpeedUpDSCount=LREAL_TO_UDINT(Time_DS*gvl.sampleRate) THEN
	SpeedUpSubState:=SpeedUpSS;
	EnterSpeedUpSPCount:=gait_cycle;
	body_ref_pos_enter :=body_ref_pos;
	body_ref_ang_enter:=body_ref_ang;
	leg_ref_pos_enter := leg_ref_pos;
	SpeedUpFinished:=TRUE;
	tipForceDesire:=tipForceDesireZeros;
	RequireSlide:=TRUE;
END_IF

body_ref_pos:=body_ref_pos_enter;
body_ref_ang:=body_ref_ang_enter;
leg_ref_pos:=leg_ref_pos_enter;

IF SpeedUpSubState=SpeedUpAS AND gait_cycle-EnterSpeedUpASCount<=Time_AS*gvl.sampleRate THEN
	fbHermitInterpolation(t0:=EnterSpeedUpASCount*delta_t , T:=Time_AS , y0:=0 , 
		y1:=Distance_x_AS , v0:=0 , v1:=target_vel , tNow:=gait_cycle* delta_t, 
		y=> body_ref_pos_wrt_body.data[0], v=>invalid );	
	body_ref_pos_wrt_body.data[1]:=0;body_ref_pos_wrt_body.data[2]:=0;
	fbRotMat(yaw := body_ref_ang_enter.data[2], pitch := body_ref_ang_enter.data[1],roll := body_ref_ang_enter.data[0], rm =>  Rb_target1 );
	body_ref_pos:=VecAdd(body_ref_pos_enter,MatMulVec(Rb_target1,body_ref_pos_wrt_body));
	
	//force compensator
	tipForceTarget:=tipForceDesireLegAF;
	IF (gait_cycle-EnterSpeedUpASCount)<=fceLoadTime*gvl.sampleRate THEN
		tr  := UDINT_TO_LREAL(gait_cycle-EnterSpeedUpASCount) / gvl.sampleRate / fceLoadTime;
		fbGetPivot(tNow := tr, tTotal := 1.0, pivot => pvt);
		FOR i:=0 TO 5 DO
			FOR j:=0 TO 2 DO
				tipForceDesire[i,j]:=(1-pvt)*tipForceDesireZeros[i,j]+pvt*tipForceTarget[i,j];
			END_FOR
		END_FOR	
	END_IF
	
END_IF
	//force compensator
	tipForceTarget:=tipForceDesireLegAF;
	IF (gait_cycle-EnterSpeedUpASCount)>(Time_AS+Time_CS-fceLoadTime)*gvl.sampleRate AND (gait_cycle-EnterSpeedUpASCount)<=(Time_AS+Time_CS)*gvl.sampleRate THEN
		tr  := (UDINT_TO_LREAL(gait_cycle-EnterSpeedUpASCount) / gvl.sampleRate- (Time_AS+Time_CS-fceLoadTime))/ fceLoadTime;
		fbGetPivot(tNow := tr, tTotal := 1.0, pivot => pvt);
		FOR i:=0 TO 5 DO
			FOR j:=0 TO 2 DO
				tipForceDesire[i,j]:=(1-pvt)*tipForceTarget[i,j]+pvt*tipForceDesireZeros[i,j];
			END_FOR
		END_FOR	
	END_IF

IF SpeedUpSubState=SpeedUpCS AND gait_cycle-EnterSpeedUpCSCount<=Time_CS*gvl.sampleRate THEN
	fbHermitInterpolation(t0:=EnterSpeedUpCSCount*delta_t , T:=Time_CS , y0:=0 , 
		y1:=target_vel*Time_CS , v0:=target_vel , v1:=target_vel , tNow:=gait_cycle* delta_t, 
		y=> body_ref_pos_wrt_body.data[0], v=>invalid );
	body_ref_pos_wrt_body.data[1]:=0;body_ref_pos_wrt_body.data[2]:=0;
	fbRotMat(yaw := body_ref_ang_enter.data[2], pitch := body_ref_ang_enter.data[1],roll := body_ref_ang_enter.data[0], rm =>  Rb_target1 );
	body_ref_pos:=VecAdd(body_ref_pos_enter,MatMulVec(Rb_target1,body_ref_pos_wrt_body));
END_IF
IF SpeedUpSubState=SpeedUpDS AND gait_cycle-EnterSpeedUpDSCount<=Time_DS*gvl.sampleRate THEN
	fbHermitInterpolation(t0:=EnterSpeedUpDSCount*delta_t , T:=Time_DS , y0:=0 , 
		y1:=Distance_x_DS , v0:=target_vel , v1:=0 , tNow:=gait_cycle* delta_t, 
		y=> body_ref_pos_wrt_body.data[0], v=>invalid );
	body_ref_pos_wrt_body.data[1]:=0;body_ref_pos_wrt_body.data[2]:=0;
	
	fbRotMat(yaw := body_ref_ang_enter.data[2], pitch := body_ref_ang_enter.data[1],roll := body_ref_ang_enter.data[0], rm =>  Rb_target1 );
	body_ref_pos:=VecAdd(body_ref_pos_enter,MatMulVec(Rb_target1,body_ref_pos_wrt_body));
	
	tr  := UDINT_TO_LREAL(gait_cycle - EnterSpeedUpDSCount) / gvl.sampleRate / Time_DS;
	fbGetPivot(tNow := tr, tTotal := 1.0, pivot => pvt);
	FOR i:=0 TO 1 DO
		leg_ref_pos[Mapping05[i]].data[2]:=(1-pvt)*leg_ref_pos_enter[Mapping05[i]].data[2]+pvt*(leg_ref_pos_enter[Mapping05[i]].data[2]+Distance_y_DS);
	END_FOR
	
END_IF
IF SpeedUpSubState=SpeedUpAS OR SpeedUpSubState=SpeedUpCS OR SpeedUpSubState=SpeedUpDS THEN
	FOR i:=0 TO 1 DO
		gvl.legCtrl[Mapping14[i]].ForwardKinetics(motorAngles:=SpeedUp_MJntRef[i].data , legIndex:=Mapping14[i] , tipPosition=>SpeedUp_MPosWrtHip[i].data );
		gvl.legCtrl[Mapping23[i]].ForwardKinetics(motorAngles:=SpeedUp_FJntRef[i].data , legIndex:=Mapping23[i] , tipPosition=>SpeedUp_FPosWrtHip[i].data );
		fbRotMat(yaw := body_ref_ang_enter.data[2], pitch := body_ref_ang_enter.data[1],roll := body_ref_ang_enter.data[0], rm =>  Rb_target1 );
		temp.data[0]:=hip_pos[Mapping14[i],0];temp.data[1]:=hip_pos[Mapping14[i],1];temp.data[2]:=hip_pos[Mapping14[i],2];
		leg_ref_pos[Mapping14[i]]:= VecAdd( MatMulVec(Rb_target1, VecAdd(temp,MatMulVec(Rleg[Mapping14[i]],SpeedUp_MPosWrtHip[i]))),body_ref_pos);
		temp.data[0]:=hip_pos[Mapping23[i],0];temp.data[1]:=hip_pos[Mapping23[i],1];temp.data[2]:=hip_pos[Mapping23[i],2];
		leg_ref_pos[Mapping23[i]]:= VecAdd( MatMulVec(Rb_target1, VecAdd(temp,MatMulVec(Rleg[Mapping23[i]],SpeedUp_FPosWrtHip[i]))),body_ref_pos);
	END_FOR
END_IF
END_METHOD

METHOD PUBLIC TrjPlanning_StoneRot : BOOL
VAR_INPUT
END_VAR
VAR
	(*StoneRot_FJntTarget:ARRAY[0..1,0..2] OF LREAL:=[-90*pi/180,524*pi/180,-190*pi/180,
                                                     90*pi/180,524*pi/180,-190*pi/180];*)
													 
	(*StoneRot_FJntTarget:ARRAY[0..1,0..2] OF LREAL:=[-90*pi/180,165*pi/180,(-190+360)*pi/180,
                                                     90*pi/180,165*pi/180,(-190+360)*pi/180];	//164 lose,165T 170S lose;*)
											 
	tr: LREAL;
	i: INT;
	Rb_target1: Mat3;	
	temp:vec3;										 
	j: INT;
	noPlanning: BOOL;
END_VAR
//*****************************test trajectory*****************************************

	FOR i:=0 TO 1 DO
		(*IF SetColide=TRUE THEN
			gvl.tipActualFce[Mapping23[i],2]:=100;
		END_IF	*)
		(*IF(gait_cycle-EnterStoneRotCount)=0.5*StoneGripTime*gvl.sampleRate THEN
			gvl.tipActualFce[Mapping23[i],2]:=100;
		END_IF *)
		noPlanning:=TRUE;
	END_FOR
	

//**********************************end************************************************	
//***********************************夹取新冰壶位置调整********* start*******************
IF gait_cycle-EnterStoneRotCount=1 THEN
	StoneRot_FJntTarget[0,1]:=gvl.gripBallThighTargetAngle*pi/180;//right leg thigh
	StoneRot_FJntTarget[1,1]:=gvl.gripBallThighTargetAngle*pi/180;//left leg thigh
	StoneRot_FJntTarget[0,2]:=gvl.gripBallShankTargetAngle*pi/180;//right leg shank
	StoneRot_FJntTarget[1,2]:=gvl.gripBallShankTargetAngle*pi/180;//left leg shank
	
END_IF
//************************************end************************************************

(*FOR i:=0 TO 1 DO
	IF StoneRotSubState[i]=FALSE AND isStone(Mapping23[i]) THEN
		StoneRotSubState[i]:=TRUE;
		leg_ref_pos_enter[Mapping23[i]]:=leg_ref_pos[Mapping23[i]];
	END_IF
END_FOR*)

IF (StoneRotSubState[0]=FALSE OR StoneRotSubState[1]=FALSE) AND (gait_cycle-EnterStoneRotCount)=LREAL_TO_UDINT(StoneGripTime*gvl.sampleRate) THEN
	StoneRotSubState[0]:=TRUE;
	StoneRotSubState[1]:=TRUE;
	leg_ref_pos_enter[Mapping23[0]]:=leg_ref_pos[Mapping23[0]];
	leg_ref_pos_enter[Mapping23[1]]:=leg_ref_pos[Mapping23[1]];
END_IF
	
body_ref_pos:=body_ref_pos_enter;
body_ref_ang:=body_ref_ang_enter;
leg_ref_pos:=leg_ref_pos_enter;


	IF (gait_cycle-EnterStoneRotCount)<=StoneGripTime*gvl.sampleRate THEN
		FOR i:=0 TO 1 DO
			IF StoneRotSubState[i]=FALSE THEN
			tr  := UDINT_TO_LREAL(gait_cycle - EnterStoneRotCount) / gvl.sampleRate /StoneGripTime;
			fbGetPivot(tNow := tr, tTotal := 1.0, pivot => pvt);
			FOR j:=0 TO 2 DO
				StoneRot_FJntRef[i].data[j]:=(1-pvt)*StoneRot_FJntStart[i].data[j]+pvt*(StoneRot_FJntTarget[i,j]);
			END_FOR
			gvl.legCtrl[Mapping23[i]].ForwardKinetics(motorAngles:=StoneRot_FJntRef[i].data , legIndex:=Mapping23[i] , tipPosition=>StoneRot_FPosWrtHip[i].data );
			fbRotMat(yaw := body_ref_ang_enter.data[2], pitch := body_ref_ang_enter.data[1],roll := body_ref_ang_enter.data[0], rm =>  Rb_target1 );
			temp.data[0]:=hip_pos[Mapping23[i],0];temp.data[1]:=hip_pos[Mapping23[i],1];temp.data[2]:=hip_pos[Mapping23[i],2];
			leg_ref_pos[Mapping23[i]]:= VecAdd( MatMulVec(Rb_target1, VecAdd(temp,MatMulVec(Rleg[Mapping23[i]],StoneRot_FPosWrtHip[i]))),body_ref_pos);
			END_IF
		END_FOR
	ELSE
		noPlanning:=TRUE;
	END_IF

IF (gait_cycle-EnterStoneRotCount)>StoneGripTime*gvl.sampleRate  THEN
		stone_rot_vel:=GVL.stone_rot_vel/60*2*pi;
		GVL.jogVelocity[18]:=stone_rot_vel;
		GVL.jogVelocity[19]:=-stone_rot_vel;
		FOR j:=18 TO 19 DO
			gvl.motorDrive[j].SetTrgVel(GVL.jogVelocity[j]);
			IF gvl.motorDrive[j].cvSetVel = GVL.jogVelocity[j] THEN
				gvl.jogButton[j]:=FALSE;
			ELSE
				gvl.jogButton[j]:=TRUE;
			END_IF
		END_FOR
END_IF

IF StoneRotFinished=FALSE AND (gait_cycle-EnterStoneRotCount)>=(StoneGripTime+StoneRotTime)*gvl.sampleRate THEN
	StoneRotFinished:=TRUE;
END_IF
END_METHOD

END_FUNCTION_BLOCK

// ---- POUs/GaitPlanner/RcToSlipFromCurling.TcPOU
FUNCTION_BLOCK RcToSlipFromCurling
VAR_INPUT
END_VAR
VAR_OUTPUT
END_VAR
VAR
//*********************************common state start*********************************************	
	gait_cycle : UDINT := 0;
	quit_flag : BOOL := FALSE;
	delta_t:LREAL:=0.001;//sampling period
	isFinished:BOOL:=FALSE;
	// robot geometrical parameters
	hip_pos : ARRAY[0..5, 0..2] OF LREAL := [-0.369,  -0.125, 0,
                                             0,  -0.28, 0,
                                             0.36, -0.125, 0,
                                             0.36, 0.125, 0,
											 0,0.28,0,
											 -0.369,0.125,0];

	leg_index_mapping : ARRAY[0..5] OF INT := [1, 2, 3, 4,5,6];
	Rleg : ARRAY[0..5] OF Mat3;
	
	joint_ref_pos_init : ARRAY[0..5] OF Vec3;
	jointPosLast   : ARRAY[0..5, 0..2] OF LREAL; 
	
	body_ref_pos_init : Vec3;
	body_ref_ang_init : Vec3;
    leg_ref_pos_init : ARRAY[0..5] OF Vec3;
	leg_ref_pos_init_wrt_hip : ARRAY[0..5] OF Vec3;
	
	body_ref_pos_enter : Vec3;
	body_ref_ang_enter : Vec3;
    leg_ref_pos_enter : ARRAY[0..5] OF Vec3;
	
	body_ref_pos : Vec3;
	body_ref_ang : Vec3;
    leg_ref_pos : ARRAY[0..5] OF Vec3;
	leg_ref_pos_wrt_hip : ARRAY[0..5] OF Vec3;
	
	body_ref_pos_next : Vec3;
	body_ref_ang_next : Vec3;
    leg_ref_pos_next : ARRAY[0..5] OF Vec3;
	leg_ref_pos_next_wrt_hip : ARRAY[0..5] OF Vec3;
	leg_ref_vel_next_wrt_hip : ARRAY[0..5] OF Vec3;
	
	// output test
	joint_ref_pos   : ARRAY[0..5] OF Vec3;
	joint_ref_vel   : ARRAY[0..5] OF Vec3;
	
	jointPosTarget  : ARRAY[0..5, 0..2] OF LREAL; 
	jointVelTarget  : ARRAY[0..5, 0..2] OF LREAL;  
	jointFceTarget  : ARRAY[0..5, 0..2] OF LREAL;  
	
	pvt, pvtDot : LREAL;
	
	fbRotmat : RotM;
	fbGetPivot  : GetPivot;
	fbCubicSpline:CubicSpline;
	
	Mapping05:ARRAY[0..1] OF INT:=[0,5];
	Mapping14:ARRAY[0..1] OF INT:=[1,4];
	Mapping23:ARRAY[0..1] OF INT:=[2,3];
//*********************************common state end*********************************************

//*********************************exclusive state start****************************************
	BJntStart:ARRAY[0..1] OF vec3;
	BPosWrtHip:ARRAY[0..1] OF vec3;
	BJntRef:ARRAY[0..1] OF vec3;
	
	BJntRetract:ARRAY[0..1,0..2] OF LREAL;
	BJntExtend:ARRAY[0..1,0..2] OF LREAL;
	BPosRetract:ARRAY[0..1,0..2] OF LREAL:=[-0.35,-0.0887,0,
                                            -0.35,-0.0887,0];
	BPosExtend:ARRAY[0..1,0..2] OF LREAL:=[-0.35,-0.1687, 0,
                                           -0.35,-0.1687, 0];
	BJntRetractRef:ARRAY[0..1,0..2] OF LREAL:=[0*pi/180,125.3866*pi/180,263.0554*pi/180,
                                            0*pi/180,125.3866*pi/180,263.0554*pi/180];

	FJntStart:ARRAY[0..1] OF vec3;
	FPosWrtHip:ARRAY[0..1] OF vec3;
	FJntRef:ARRAY[0..1] OF vec3;	
	FJntGrip:ARRAY[0..1,0..2] OF LREAL:=[-90*pi/180,(522-360)*pi/180,(-188+360)*pi/180,
                                        90*pi/180,(522-360)*pi/180,(-188+360)*pi/180];		
	MJntStart:ARRAY[0..1] OF vec3;
	MPosWrtHip:ARRAY[0..1] OF vec3;
	MJntRef:ARRAY[0..1] OF vec3;	
	
	MJntLiftTarget:ARRAY[0..1,0..2] OF LREAL;
	MPosLiftTarget:ARRAY[0..1,0..2] OF LREAL:=[-0.0141,-0.1797+0.05,-0.1246,
                                               -0.0141,-0.1797+0.05,0.1246];
	MJntLiftTargetRef:ARRAY[0..1,0..2] OF LREAL:=[0,331.45*pi/180,-149*pi/180,
                                               0,331.45*pi/180,-149*pi/180];	
	BRetractTime:LREAL:=4;
	BExtendTime:LREAL:=2;
	FGripTime:LREAL:=2;		
	MLiftTime:LREAL:=2;	
	
	isBMove: BOOL:=FALSE;	
	isMMove: BOOL:=FALSE;	
	isFMove: BOOL:=FALSE;	
	enterMMoveCount:UDINT;	
	enterFMoveCount:UDINT;			
//*********************************exclusive state end****************************************
END_VAR

METHOD PUBLIC DoPlanning : BOOL
VAR_INPUT
	count : UDINT;
END_VAR
VAR
	i, j  : INT;
	tempLeg:ARRAY [0..2] OF LREAL;
	tempJnt:ARRAY [0..2] OF LREAL;
	tempRef:ARRAY [0..2] OF LREAL;
END_VAR
IF count = 0 THEN
	isFinished := FALSE;
	Initialize();
	FOR i:=0 TO 1 DO
		tempLeg[0]:=BPosExtend[i,0];tempLeg[1]:=BPosExtend[i,1];tempLeg[2]:=BPosExtend[i,2];
		tempRef[0]:=BJntRetractRef[i,0];tempRef[1]:=BJntRetractRef[i,1];tempRef[2]:=BJntRetractRef[i,2];
		GVL.legCtrl[Mapping05[i]].InverseKinetics(tipPosition:=tempLeg , refPosLast:=tempRef , legIndex:=Mapping05[i] , motorAngles=>tempJnt , isSingular=> );
		BJntExtend[i,0]:=tempJnt[0];BJntExtend[i,1]:=tempJnt[1];BJntExtend[i,2]:=tempJnt[2];
	END_FOR	
	FOR i:=0 TO 1 DO
		tempLeg[0]:=BPosRetract[i,0];tempLeg[1]:=BPosRetract[i,1];tempLeg[2]:=BPosRetract[i,2];
		tempRef[0]:=BJntRetractRef[i,0];tempRef[1]:=BJntRetractRef[i,1];tempRef[2]:=BJntRetractRef[i,2];
		GVL.legCtrl[Mapping05[i]].InverseKinetics(tipPosition:=tempLeg , refPosLast:=tempRef , legIndex:=Mapping05[i] , motorAngles=>tempJnt , isSingular=> );
		BJntRetract[i,0]:=tempJnt[0];BJntRetract[i,1]:=tempJnt[1];BJntRetract[i,2]:=tempJnt[2];
	END_FOR	
	FOR i:=0 TO 1 DO
		tempLeg[0]:=MPosLiftTarget[i,0];tempLeg[1]:=MPosLiftTarget[i,1];tempLeg[2]:=MPosLiftTarget[i,2];
		tempRef[0]:=MJntLiftTargetRef[i,0];tempRef[1]:=MJntLiftTargetRef[i,1];tempRef[2]:=MJntLiftTargetRef[i,2];
		GVL.legCtrl[Mapping14[i]].InverseKinetics(tipPosition:=tempLeg , refPosLast:=tempRef , legIndex:=Mapping14[i] , motorAngles=>tempJnt , isSingular=> );
		MJntLiftTarget[i,0]:=tempJnt[0];MJntLiftTarget[i,1]:=tempJnt[1];MJntLiftTarget[i,2]:=tempJnt[2];
	END_FOR		
END_IF

TrjPlanning();

IF quit_flag THEN
	isFinished := TRUE;
	quit_flag := FALSE;
END_IF
END_METHOD

METHOD PUBLIC Initialize : BOOL
VAR_INPUT
END_VAR
VAR
	i, j : INT;
	sum_height : LREAL := 0;
	leg_pos    : ARRAY[0..2] OF LREAL;
	
	Rb : Mat3;
	hip_pos_j  : Vec3;
	leg_pos_wrt_com : Vec3;
	
END_VAR
Rleg[0]:=SetMat3(1,0,0,0,0,-1,0,1,0);
Rleg[1]:=SetMat3(-1,0,0,0,0,1,0,1,0,);
Rleg[2]:=SetMat3(-1,0,0,0,0,1,0,1,0);
Rleg[3]:=SetMat3(-1,0,0,0,0,1,0,1,0);
Rleg[4]:=SetMat3( -1,0,0,0,0,1,0,1,0);
Rleg[5]:=SetMat3(1,0,0,0,0,-1,0,1,0);

quit_flag  := FALSE;
gait_cycle := 0;
isBMove:=TRUE;
isMMove:=FALSE;
isFMove:=FALSE;
delta_t:=1.0/gvl.sampleRate;

FOR i := 0 TO 5 DO
	FOR j := 0 TO 2 DO
		IF ABS(gvl.jntLastRefPos[i, j] - gvl.jntActualPos[i, j]) < 0.2 THEN
			joint_ref_pos_init[i].data[j] := gvl.jntLastRefPos[i, j];
		ELSE
			joint_ref_pos_init[i].data[j] := gvl.jntActualPos[i, j];
		END_IF
		jointPosLast[i,j]:=joint_ref_pos_init[i].data[j];
	END_FOR
END_FOR

sum_height := 0;
FOR j := 0 TO 5 DO
	// FK
	gvl.legCtrl[j].ForwardKinetics(motorAngles := joint_ref_pos_init[j].data, legIndex:=j, tipPosition => leg_pos);
	leg_ref_pos_init_wrt_hip[j] := SetVec3(leg_pos[0], leg_pos[1], leg_pos[2]);
	sum_height := sum_height - leg_ref_pos_init_wrt_hip[j].data[1];
END_FOR
body_ref_pos_init := SetVec3(0, 0, sum_height/6.0);
body_ref_ang_init := SetVec3(0, 0, 0);                            

FOR j := 0 TO 5 DO
	fbRotMat(yaw := body_ref_ang_init.data[2],
             pitch := body_ref_ang_init.data[1],
             roll := body_ref_ang_init.data[0],
             rm => Rb );
	hip_pos_j := SetVec3(hip_pos[j, 0], hip_pos[j, 1], hip_pos[j, 2]);
	leg_pos_wrt_com := VecAdd(MatMulVec(Rleg[j], leg_ref_pos_init_wrt_hip[j]), hip_pos_j);
    leg_ref_pos_init[j] := VecAdd(body_ref_pos_init, MatMulVec(Rb, leg_pos_wrt_com));
END_FOR

body_ref_pos := body_ref_pos_init;
body_ref_ang := body_ref_ang_init;
leg_ref_pos := leg_ref_pos_init;
leg_ref_pos_wrt_hip := leg_ref_pos_init_wrt_hip;

body_ref_pos_enter := body_ref_pos_init;
body_ref_ang_enter := body_ref_ang_init;
leg_ref_pos_enter := leg_ref_pos_init;

FOR i:=0 TO 1 DO
	FOR j:=0 TO 2 DO
		BJntStart[i].data[j]:=joint_ref_pos_init[Mapping05[i]].data[j];
		MJntStart[i].data[j]:=joint_ref_pos_init[Mapping14[i]].data[j];
		FJntStart[i].data[j]:=joint_ref_pos_init[Mapping23[i]].data[j];
	END_FOR
END_FOR

FOR i := 0 TO 5 DO
	FOR j := 0 TO 2 DO
		jointPosTarget[i, j] := joint_ref_pos_init[i].data[j];
		jointVelTarget[i, j] := 0;
		jointFceTarget[i, j] := 0;
	END_FOR
END_FOR
END_METHOD

METHOD PUBLIC TrjPlanning : BOOL
VAR_INPUT
END_VAR

VAR
	tr: lreal;
	i: INT;
	j: INT;
	Rb_target1: Mat3;
	temp: vec3;
	
	Rb: Mat3;
	hip_pos_j: Vec3;
	leg_ref_pos_wrt_com_j: Vec3;
	tmp: Vec3;
	tip_pos: Vec3;
	tip_vel: Vec3;
	jointTmpPosLast: ARRAY [0..2] OF LREAL;
END_VAR
gait_cycle := gait_cycle + 1;

IF gait_cycle=LREAL_TO_UDINT((BRetractTime+BExtendTime)*gvl.sampleRate) OR (gait_cycle-enterMMoveCount) =LREAL_TO_UDINT(MLiftTime*gvl.sampleRate) OR (gait_cycle-enterFMoveCount)=LREAL_TO_UDINT(FGripTime*gvl.sampleRate) THEN
	leg_ref_pos_enter:=leg_ref_pos;
END_IF

IF isMMove=FALSE AND isFMove=FALSE THEN
IF isBMove=TRUE THEN
	body_ref_pos:=body_ref_pos_enter;
	body_ref_ang:=body_ref_ang_enter;
	leg_ref_pos:=leg_ref_pos_enter;
	IF gait_cycle<=BRetractTime*gvl.sampleRate  THEN
		tr  := UDINT_TO_LREAL(gait_cycle) / gvl.sampleRate /BRetractTime;
		fbGetPivot(tNow := tr, tTotal := 1.0, pivot => pvt);
		FOR i:=0 TO 1 DO
			FOR j:=0 TO 2 DO
				BJntRef[i].data[j]:=(1-pvt)*BJntStart[i].data[j]+pvt*(BJntRetract[i,j]);
			END_FOR
			gvl.legCtrl[Mapping05[i]].ForwardKinetics(motorAngles:=BJntRef[i].data , legIndex:=Mapping05[i] , tipPosition=>BPosWrtHip[i].data );
			fbRotMat(yaw := body_ref_ang_init.data[2], pitch := body_ref_ang_init.data[1],roll := body_ref_ang_init.data[0], rm =>  Rb_target1 );
			temp.data[0]:=hip_pos[Mapping05[i],0];temp.data[1]:=hip_pos[Mapping05[i],1];temp.data[2]:=hip_pos[Mapping05[i],2];
			leg_ref_pos[Mapping05[i]]:= VecAdd( MatMulVec(Rb_target1, VecAdd(temp,MatMulVec(Rleg[Mapping05[i]],BPosWrtHip[i]))),body_ref_pos);
		END_FOR
	ELSIF gait_cycle<=(BRetractTime+BExtendTime)*gvl.sampleRate THEN
		tr  := (UDINT_TO_LREAL(gait_cycle) / gvl.sampleRate- BRetractTime)/BExtendTime;
		fbGetPivot(tNow := tr, tTotal := 1.0, pivot => pvt);
		FOR i:=0 TO 1 DO
			FOR j:=0 TO 2 DO
				BJntRef[i].data[j]:=(1-pvt)*BJntRetract[i,j]+pvt*BJntExtend[i,j];
			END_FOR
			gvl.legCtrl[Mapping05[i]].ForwardKinetics(motorAngles:=BJntRef[i].data , legIndex:=Mapping05[i] , tipPosition=>BPosWrtHip[i].data );
			fbRotMat(yaw := body_ref_ang_init.data[2], pitch := body_ref_ang_init.data[1],roll := body_ref_ang_init.data[0], rm =>  Rb_target1 );
			temp.data[0]:=hip_pos[Mapping05[i],0];temp.data[1]:=hip_pos[Mapping05[i],1];temp.data[2]:=hip_pos[Mapping05[i],2];
			leg_ref_pos[Mapping05[i]]:= VecAdd( MatMulVec(Rb_target1, VecAdd(temp,MatMulVec(Rleg[Mapping05[i]],BPosWrtHip[i]))),body_ref_pos);
		END_FOR
	ELSE
		isBMove:=FALSE;
		isMMove:=TRUE;
		leg_ref_pos_enter:=leg_ref_pos;
		enterMMoveCount:=gait_cycle;
	END_IF
END_IF
END_IF

IF isBMove=FALSE AND isFMove=FALSE THEN
IF isMMove=TRUE THEN
	body_ref_pos:=body_ref_pos_enter;
	body_ref_ang:=body_ref_ang_enter;
	leg_ref_pos:=leg_ref_pos_enter;
	IF (gait_cycle-enterMMoveCount) <=MLiftTime*gvl.sampleRate THEN
		tr  := UDINT_TO_LREAL(gait_cycle- enterMMoveCount) / gvl.sampleRate/MLiftTime;
		fbGetPivot(tNow := tr, tTotal := 1.0, pivot => pvt);
		FOR i:=0 TO 1 DO
			FOR j:=0 TO 2 DO	
				MJntRef[i].data[j]:=(1-pvt)*MJntStart[i].data[j]+pvt*(MJntLiftTarget[i,j]);
			END_FOR
			gvl.legCtrl[Mapping14[i]].ForwardKinetics(motorAngles:=MJntRef[i].data , legIndex:=Mapping14[i] , tipPosition=>MPosWrtHip[i].data );
			fbRotMat(yaw := body_ref_ang_init.data[2], pitch := body_ref_ang_init.data[1],roll := body_ref_ang_init.data[0], rm =>  Rb_target1 );
			temp.data[0]:=hip_pos[Mapping14[i],0];temp.data[1]:=hip_pos[Mapping14[i],1];temp.data[2]:=hip_pos[Mapping14[i],2];
			leg_ref_pos[Mapping14[i]]:= VecAdd( MatMulVec(Rb_target1, VecAdd(temp,MatMulVec(Rleg[Mapping14[i]],MPosWrtHip[i]))),body_ref_pos);
		END_FOR
	ELSE
		isMMove:=FALSE;
		isFMove:=TRUE;
		leg_ref_pos_enter:=leg_ref_pos;
		enterFMoveCount:=gait_cycle;
	END_IF
END_IF
END_IF

IF isBMove=FALSE AND isMMove=FALSE THEN
IF isFMove=TRUE THEN
	body_ref_pos:=body_ref_pos_enter;
	body_ref_ang:=body_ref_ang_enter;
	leg_ref_pos:=leg_ref_pos_enter;
	IF (gait_cycle-enterFMoveCount) <=FGripTime*gvl.sampleRate THEN
		tr  := UDINT_TO_LREAL(gait_cycle- enterFMoveCount) / gvl.sampleRate/FGripTime;
		fbGetPivot(tNow := tr, tTotal := 1.0, pivot => pvt);
		FOR i:=0 TO 1 DO
			FOR j:=0 TO 2 DO	
				FJntRef[i].data[j]:=(1-pvt)*FJntStart[i].data[j]+pvt*(FJntGrip[i,j]);
			END_FOR
		gvl.legCtrl[Mapping23[i]].ForwardKinetics(motorAngles:=FJntRef[i].data , legIndex:=Mapping23[i] , tipPosition=>FPosWrtHip[i].data );
		fbRotMat(yaw := body_ref_ang_init.data[2], pitch := body_ref_ang_init.data[1],roll := body_ref_ang_init.data[0], rm =>  Rb_target1 );
		temp.data[0]:=hip_pos[Mapping23[i],0];temp.data[1]:=hip_pos[Mapping23[i],1];temp.data[2]:=hip_pos[Mapping23[i],2];
		leg_ref_pos[Mapping23[i]]:= VecAdd( MatMulVec(Rb_target1, VecAdd(temp,MatMulVec(Rleg[Mapping23[i]],FPosWrtHip[i]))),body_ref_pos);
		END_FOR
	ELSE
		isFMove:=FALSE;
		leg_ref_pos_enter:=leg_ref_pos;
		isFinished := TRUE;
	END_IF
END_IF
END_IF

// transform TO leg local frame AND DO inverse kinematics
FOR j := 0 TO 5 DO
	fbRotMat(
    	yaw := body_ref_ang.data[2], 
		pitch := body_ref_ang.data[1], 
		roll := body_ref_ang.data[0], 
		rm => Rb);
	hip_pos_j := SetVec3(hip_pos[j, 0], hip_pos[j, 1], hip_pos[j, 2]);

	//leg_ref_pos_wrt_com = Rb' * (leg_ref_pos - body_ref_pos)
	leg_ref_pos_wrt_com_j := MatMulVec(
		                         MatTranspose(Rb),
								 VecAdd(
									 leg_ref_pos[j],
									 VecNeg(body_ref_pos)
                                 )
                             );
	// leg_ref_pos_wrt_hip = Rleg' * (leg_ref_pos_wrt_com_j - hip_pos)
	leg_ref_pos_next_wrt_hip[j] := MatMulVec(
		                               MatTranspose(Rleg[j]),
									   VecAdd(
										   leg_ref_pos_wrt_com_j,
										   VecNeg(hip_pos_j)
									   )
								   );
								   
	leg_ref_vel_next_wrt_hip[j] := VecMulNum(VecAdd(leg_ref_pos_next_wrt_hip[j], VecNeg(leg_ref_pos_wrt_hip[j])), DINT_TO_LREAL(gvl.sampleRate));
END_FOR


// mapping to actual joints
FOR j := 0 TO 5 DO
	tmp := leg_ref_pos_next_wrt_hip[leg_index_mapping[j]-1];
	tip_pos := SetVec3(tmp.data[0], tmp.data[1], tmp.data[2]);
	tmp := leg_ref_vel_next_wrt_hip[leg_index_mapping[j]-1];
	tip_vel := SetVec3(tmp.data[0], tmp.data[1], tmp.data[2]);
	FOR i:= 0 TO 2 DO
		jointTmpPosLast[i]:=jointPosLast[j,i];
	END_FOR		
	gvl.legCtrl[j].InversePosAndVel(
		tipPos := tip_pos.data, 
		tipVel := tip_vel.data, 
		refPosLast:=jointTmpPosLast,
		legIndex:=j,
		jntPos => joint_ref_pos[j].data, 
		jntVel => joint_ref_vel[j].data);
	
END_FOR

// link to physical outputs
FOR i := 0 TO 5 DO
	FOR j := 0 TO 2 DO
		jointPosTarget[i, j] := joint_ref_pos[i].data[j];
		jointPosLast[i,j]:=jointPosTarget[i, j] ;
		jointVelTarget[i, j] := joint_ref_vel[i].data[j];
		jointFceTarget[i, j] := 0;
	END_FOR
END_FOR

// store refs for next loop
leg_ref_pos_wrt_hip := leg_ref_pos_next_wrt_hip;
END_METHOD

END_FUNCTION_BLOCK

// ---- POUs/tools/CubicSpline.TcPOU
FUNCTION_BLOCK CubicSpline//参考《数值分析》第4版李庆扬等编，p36三转角方程
VAR_INPUT
	x : ARRAY[0..4] OF LREAL;
	y : ARRAY[0..4] OF LREAL;
	dy0 : LREAL;
	dy4 : LREAL;
	xt: LREAL;
END_VAR
VAR_OUTPUT
	yt: LREAL;
	vt: LREAL;
END_VAR
VAR
	i : INT;
	h : ARRAY[0..3] OF LREAL;
	f : ARRAY[0..3] OF LREAL;
	lemda : ARRAY[0..3] OF LREAL;
	miu : ARRAY[0..3] OF LREAL;
	g : ARRAY[0..3] OF LREAL;

	//lftMat*lftVec=rghtVec，求lftVec
	lftMat : Mat3;
	lftVec : Vec3;
	rghtVec : Vec3;
	m: ARRAY[0..4] OF LREAL;
	alpha: ARRAY[0..4] OF LREAL;
	beta: ARRAY[0..4] OF LREAL;
	dAlpha: ARRAY[0..4] OF LREAL;
	dBeta: ARRAY[0..4] OF LREAL;
	tmp: LREAL;
	tmpd: LREAL;
END_VAR

FOR i:=0 TO 3 DO
	h[i] := x[i+1] - x[i];
	f[i] := (y[i+1] - y[i]) / h[i];
END_FOR

FOR i:=1 TO 3 DO
	lemda[i] := h[i] / (h[i-1] + h[i]);
	miu[i] := h[i-1] / (h[i-1] + h[i]);
	g[i] := 3 * (lemda[i] * f[i-1] + miu[i] * f[i]);
END_FOR

//才3*3，直接求逆，更大的矩阵用追赶法
lftMat := SetMat3(2,miu[1],0, lemda[2],2,miu[2], 0,lemda[3],2);
rghtVec := SetVec3(g[1]-lemda[1]*dy0, g[2], g[3]-miu[3]*dy4);
lftVec := MatMulVec(Inv3(lftMat), rghtVec);
m[0] := dy0;
FOR i:=0 TO 2 DO
	m[i+1] := lftVec.data[i];
END_FOR
m[4] := dy4;

//分段三次hermite插值
i:=0;
IF xt <= x[1] THEN//i=0
	tmp := (xt-x[i+1])/(x[i]-x[i+1]) * (xt-x[i+1])/(x[i]-x[i+1]);
	alpha[i] := tmp * (1+2*(xt-x[i])/(x[i+1]-x[i]));
	beta[i]  := tmp * (xt-x[i]);
	tmpd := (xt-x[i+1])/(x[i]-x[i+1])/(x[i]-x[i+1]);
	dAlpha[i] := tmpd * 6*(xt-x[i])/(x[i+1]-x[i]);
	dBeta[i]  := tmpd * (2*(xt-x[i])+(xt-x[i+1]));
ELSE
	alpha[i] := 0;
	beta[i]  := 0;
	dAlpha[i]:= 0;
	dBeta[i] := 0;
END_IF
FOR i:=1 TO 3 DO
	IF xt >= x[i-1] AND xt <= x[i] THEN
		tmp := (xt-x[i-1])/(x[i]-x[i-1]) * (xt-x[i-1])/(x[i]-x[i-1]);
		alpha[i] := tmp * (1+2*(xt-x[i])/(x[i-1]-x[i]));
		beta[i]  := tmp * (xt-x[i]);
		tmpd := (xt-x[i-1])/(x[i]-x[i-1])/(x[i]-x[i-1]);
		dAlpha[i] := tmpd * 6*(xt-x[i])/(x[i-1]-x[i]);
		dBeta[i]  := tmpd * (2*(xt-x[i])+(xt-x[i-1]));
	ELSIF xt >= x[i] AND xt <= x[i+1] THEN
		tmp := (xt-x[i+1])/(x[i]-x[i+1]) * (xt-x[i+1])/(x[i]-x[i+1]);
		alpha[i] := tmp * (1+2*(xt-x[i])/(x[i+1]-x[i]));
		beta[i]  := tmp * (xt-x[i]);
		tmpd := (xt-x[i+1])/(x[i]-x[i+1])/(x[i]-x[i+1]);
		dAlpha[i] := tmpd * 6*(xt-x[i])/(x[i+1]-x[i]);
		dBeta[i]  := tmpd * (2*(xt-x[i])+(xt-x[i+1]));
	ELSE
		alpha[i] := 0;
		beta[i]  := 0;
		dAlpha[i]:= 0;
		dBeta[i] := 0;
	END_IF
END_FOR
i:=4;
IF xt >= x[3] THEN
	tmp := (xt-x[i-1])/(x[i]-x[i-1]) * (xt-x[i-1])/(x[i]-x[i-1]);
	alpha[i] := tmp * (1+2*(xt-x[i])/(x[i-1]-x[i]));
	beta[i]  := tmp * (xt-x[i]);
	tmpd := (xt-x[i-1])/(x[i]-x[i-1])/(x[i]-x[i-1]);
	dAlpha[i] := tmpd * 6*(xt-x[i])/(x[i-1]-x[i]);
	dBeta[i]  := tmpd * (2*(xt-x[i])+(xt-x[i-1]));
ELSE
	alpha[i] := 0;
	beta[i]  := 0;
	dAlpha[i]:= 0;
	dBeta[i] := 0;
END_IF

yt:=0;
vt:=0;
FOR i:=0 TO 4 DO
	yt := yt + y[i]*alpha[i] + m[i]*beta[i];
	vt := vt + y[i]*dAlpha[i] + m[i]*dBeta[i];
END_FOR

END_FUNCTION_BLOCK

// ---- POUs/tools/VectorMath/Inv3.TcPOU
FUNCTION Inv3 : Mat3
VAR_INPUT
	A : Mat3;
END_VAR
VAR
	a1, a2, a3, b1, b2, b3, c1, c2, c3 : LREAL;
	detA : LREAL;
END_VAR

a1 := A.data[0, 0]; a2 := A.data[0, 1]; a3 := A.data[0, 2];
b1 := A.data[1, 0]; b2 := A.data[1, 1]; b3 := A.data[1, 2];
c1 := A.data[2, 0]; c2 := A.data[2, 1]; c3 := A.data[2, 2];

detA := -a3 * b2 * c1 + a2 * b3 * c1 + a3 * b1 * c2 - a1 * b3 * c2 - a2 * b1 * c3 + a1 * b2 * c3;

IF ABS(detA) < 1E-12 THEN
	// avoid singularity, leave other things to user
	detA := 1E-12;
END_IF

Inv3.data[0, 0] := ( -b3 * c2 + b2 * c3 ) / detA; Inv3.data[0, 1] := ( a3 * c2 - a2 * c3 ) / detA; Inv3.data[0, 2] := ( -a3 * b2 + a2 * b3 ) / detA;
Inv3.data[1, 0] := (  b3 * c1 - b1 * c3 ) / detA; Inv3.data[1, 1] := (-a3 * c1 + a1 * c3 ) / detA; Inv3.data[1, 2] := (  a3 * b1 - a1 * b3 ) / detA;
Inv3.data[2, 0] := ( -b2 * c1 + b1 * c2 ) / detA; Inv3.data[2, 1] := ( a2 * c1 - a1 * c2 ) / detA; Inv3.data[2, 2] := ( -a2 * b1 + a1 * b2 ) / detA;

END_FUNCTION

// ---- POUs/GaitPlanner/BLegSlip.TcPOU
FUNCTION_BLOCK BLegSlip
VAR_INPUT
END_VAR
VAR_OUTPUT
END_VAR
VAR
	period:LREAL:=1;//total time of swing and stance
	duty:LREAL:=0.5;
	step_height:LREAL:=0.08;
	step:ARRAY [0..2] OF LREAL:=[0.1,0.1,0.1];//velocity change step
	delta_t:LREAL:=0.001;//sampling period
	
	// robot geometrical parameters
	hip_pos : ARRAY[0..5, 0..2] OF LREAL := [-0.369,  -0.125, 0,
                                             0,  -0.28, 0,
                                             0.36, -0.125, 0,
                                             0.36, 0.125, 0,
											 0,0.28,0,
											 -0.369,0.125,0];

	leg_index_mapping : ARRAY[0..5] OF INT := [1, 2, 3, 4,5,6];
	Rleg : ARRAY[0..5] OF Mat3;
	
	joint_ref_pos_init : ARRAY[0..5] OF Vec3;
	jointPosLast   : ARRAY[0..5, 0..2] OF LREAL; 
	
	body_ref_pos_init : Vec3;
	body_ref_ang_init : Vec3;
    leg_ref_pos_init : ARRAY[0..5] OF Vec3;
	leg_ref_pos_init_wrt_hip : ARRAY[0..5] OF Vec3;
	
	body_ref_pos : Vec3;
	body_ref_ang : Vec3;
    leg_ref_pos : ARRAY[0..5] OF Vec3;
	leg_ref_pos_wrt_hip : ARRAY[0..5] OF Vec3;
	
	body_ref_pos_next : Vec3;
	body_ref_ang_next : Vec3;
    leg_ref_pos_next : ARRAY[0..5] OF Vec3;
	leg_ref_pos_next_wrt_hip : ARRAY[0..5] OF Vec3;
	leg_ref_vel_next_wrt_hip : ARRAY[0..5] OF Vec3;
	
	// output test
	joint_ref_pos   : ARRAY[0..5] OF Vec3;
	joint_ref_vel   : ARRAY[0..5] OF Vec3;
	
	jointPosTarget  : ARRAY[0..5, 0..2] OF LREAL; 
	jointVelTarget  : ARRAY[0..5, 0..2] OF LREAL;  
	jointFceTarget  : ARRAY[0..5, 0..2] OF LREAL;  
	
	pvt, pvtDot : LREAL;
	
	fbRotmat : RotM;
	fbGetPivot  : GetPivot;
	fbCubicSpline:CubicSpline;
	
	//state
	stance:INT:=1;
	swing:INT:=0;
	ready:INT:=-1;
	init:INT:=-2;
	state:INT:=-1;
	state_last:INT:=-1;
	
	gait_cycle : UDINT := 0;
	gait_cycle_enter: UDINT := 0;
	quit_flag : BOOL := FALSE;
	requir_stop:BOOL:=FALSE;
	require_move_last:BOOL:=FALSE;
	require_move:BOOL:=FALSE;
	isFinished:BOOL:=FALSE;
	inSlip: BOOL:=FALSE;
	
	count_en_ST:UDINT:=0;
	count_en_SW:UDINT:=0;
	count_en_RD:UDINT:=0;
	tip_pos_en_ST:ARRAY [0..1] OF vec3;
	tip_pos_en_SW:ARRAY [0..1] OF vec3;
	tip_pos_en_RD:ARRAY [0..1] OF vec3;
	tip_vel_en_ST:ARRAY [0..1] OF vec3;
	tip_vel_en_SW:ARRAY [0..1] OF vec3;
	tip_vel_en_RD:ARRAY [0..1] OF vec3;
	tip_pos_ref:ARRAY [0..1] OF vec3;
	tip_vel_ref:ARRAY [0..1] OF vec3;
	tip_pos_ref_last:ARRAY [0..1] OF vec3;
	
	trot_vel_desire:LREAL:=0;
	side_vel_desire:LREAL:=0;
	turn_rate_desire:LREAL:=0;
	
	trot_vel:LREAL:=0;
	side_vel:LREAL:=0;
	turn_rate:LREAL:=0;
	
	trot_vel_now:LREAL:=0;
	side_vel_now:LREAL:=0;
	turn_vel_now:LREAL:=0;
	
	SwingTrj_tn:ARRAY[0..4] OF LREAL:=[0,0.25,0.5,0.75,1];
	StanceTrj_tn:ARRAY[0..4] OF LREAL:=[0,0.25,0.5,0.75,1];
	ReadyTrj_tn:ARRAY[0..4] OF LREAL:=[0,0.25,0.5,0.75,1];
	
	normal_tip_pos_cart:ARRAY[0..2] OF LREAL:=[-0.35,-0.1687,0];
	base_height:LREAL;
	base_x:LREAL;
	base_z:LREAL;
	step_height_now:LREAL;
	step_length_now:LREAL;
	step_side_len_now:LREAL;
	start_height:LREAL;
	Mapping05:ARRAY[0..1] OF INT:=[0,5];
	
END_VAR

METHOD PUBLIC Cmd2Tgt1Step : lreal
VAR_INPUT
	cmdVel:LREAL;//desired velocity
	curVel:LREAL;//current velocity
	step:LREAL;
END_VAR
VAR_OUTPUT
	trgVel:lreal;
END_VAR
IF step<0 THEN
	step:=-step;
END_IF
IF (curVel-cmdVel)<=-step THEN
    trgVel:=curVel+step;
ELSIF (curVel-cmdVel)>step THEN
    trgVel:=curVel-step;
else
    trgVel:=cmdVel;
END_IF
END_METHOD

METHOD PUBLIC DoPlanning : BOOL
VAR_INPUT
	count : UDINT;
END_VAR
VAR
	i, j  : INT;
END_VAR
IF count = 0 THEN
	isFinished := FALSE;
	Initialize();
END_IF
StateMachine();

TrjPlanning();

IF quit_flag THEN
	isFinished := TRUE;
	quit_flag := FALSE;
	inSlip:=FALSE;
	gvl.BLegSlip_trot_vel_desire:=0;
	gvl.BLegSlip_side_vel_desire:=0;
	gvl.BLegSlip_turn_rate_desire:=0;
	trot_vel_desire:=0;
	side_vel_desire:=0;
	turn_rate_desire:=0;	
END_IF
END_METHOD

METHOD PUBLIC Initialize : BOOL
VAR_INPUT
END_VAR
VAR
	i, j : INT;
	sum_height : LREAL := 0;
	leg_pos    : ARRAY[0..2] OF LREAL;
	
	Rb : Mat3;
	hip_pos_j  : Vec3;
	leg_pos_wrt_com : Vec3;
	
END_VAR
Rleg[0]:=SetMat3(1,0,0,0,0,-1,0,1,0);
Rleg[1]:=SetMat3(-1,0,0,0,0,1,0,1,0,);
Rleg[2]:=SetMat3(-1,0,0,0,0,1,0,1,0);
Rleg[3]:=SetMat3(-1,0,0,0,0,1,0,1,0);
Rleg[4]:=SetMat3( -1,0,0,0,0,1,0,1,0);
Rleg[5]:=SetMat3(1,0,0,0,0,-1,0,1,0);

quit_flag  := FALSE;
gait_cycle := 0;
state:=ready;
state_last:=init;
require_move:=FALSE;
require_move_last:=FALSE;
requir_stop:=FALSE;

FOR i := 0 TO 5 DO
	FOR j := 0 TO 2 DO
		IF ABS(gvl.jntLastRefPos[i, j] - gvl.jntActualPos[i, j]) < gvl.lift_threshold_value THEN
			joint_ref_pos_init[i].data[j] := gvl.jntLastRefPos[i, j];
		ELSE
			joint_ref_pos_init[i].data[j] := gvl.jntActualPos[i, j];
		END_IF
		jointPosLast[i,j]:=joint_ref_pos_init[i].data[j];
	END_FOR
END_FOR

sum_height := 0;
FOR j := 0 TO 5 DO
	// FK
	gvl.legCtrl[j].ForwardKinetics(motorAngles := joint_ref_pos_init[j].data, legIndex:=j, tipPosition => leg_pos);
	leg_ref_pos_init_wrt_hip[j] := SetVec3(leg_pos[0], leg_pos[1], leg_pos[2]);
	sum_height := sum_height - leg_ref_pos_init_wrt_hip[j].data[1];
END_FOR
body_ref_pos_init := SetVec3(0, 0, sum_height/6.0);
body_ref_ang_init := SetVec3(0, 0, 0);                            

FOR j := 0 TO 5 DO
	fbRotMat(yaw := body_ref_ang_init.data[2],
             pitch := body_ref_ang_init.data[1],
             roll := body_ref_ang_init.data[0],
             rm => Rb );
	hip_pos_j := SetVec3(hip_pos[j, 0], hip_pos[j, 1], hip_pos[j, 2]);
	leg_pos_wrt_com := VecAdd(MatMulVec(Rleg[j], leg_ref_pos_init_wrt_hip[j]), hip_pos_j);
    leg_ref_pos_init[j] := VecAdd(body_ref_pos_init, MatMulVec(Rb, leg_pos_wrt_com));
END_FOR

tip_pos_ref[0]:=leg_ref_pos_init_wrt_hip[Mapping05[0]];
tip_pos_ref[1]:=leg_ref_pos_init_wrt_hip[Mapping05[1]];
tip_vel_ref[0]:=setVec3(0,0,0);
tip_vel_ref[1]:=setVec3(0,0,0);
tip_pos_ref_last:=tip_pos_ref;

body_ref_pos := body_ref_pos_init;
body_ref_ang := body_ref_ang_init;
leg_ref_pos := leg_ref_pos_init;
leg_ref_pos_wrt_hip := leg_ref_pos_init_wrt_hip;

FOR i := 0 TO 5 DO
	FOR j := 0 TO 2 DO
		jointPosTarget[i, j] := joint_ref_pos_init[i].data[j];
		jointVelTarget[i, j] := 0;
		jointFceTarget[i, j] := 0;
	END_FOR
END_FOR
END_METHOD

METHOD PUBLIC StateMachine : BOOL
VAR_INPUT
END_VAR
VAR
	temp:LREAL;
	
END_VAR
//set target value
trot_vel_desire:=gvl.BLegSlip_trot_vel_desire;
side_vel_desire:=gvl.BLegSlip_side_vel_desire;
turn_rate_desire:=gvl.BLegSlip_turn_rate_desire;
step[0]:=gvl.BLegSlip_step[0];
step[1]:=gvl.BLegSlip_step[1];
step[2]:=gvl.BLegSlip_step[2];

//state switch
IF require_move_last=FALSE AND require_move=TRUE THEN
	gait_cycle_enter:=gait_cycle;
	require_move:=FALSE;
	inSlip:=TRUE;
END_IF
IF inSlip=TRUE THEN
	temp:=(gait_cycle-gait_cycle_enter) MOD TRUNC(period*gvl.sampleRate);
	IF temp>=(1-duty)*gvl.sampleRate*period THEN
		state:=stance;
	ELSE 
		state:=swing;
	END_IF
END_IF

IF state<> state_last THEN
	IF state=stance THEN
		count_en_ST:=gait_cycle;
		tip_pos_en_ST:=tip_pos_ref;
		tip_vel_en_ST:=tip_vel_ref;
	END_IF
	IF state=swing THEN
		count_en_SW:=gait_cycle;
		tip_pos_en_SW:=tip_pos_ref;
		tip_vel_en_SW:=tip_vel_ref;	
		IF requir_stop=TRUE THEN
			trot_vel_desire:=0;
			side_vel_desire:=0;
			turn_rate_desire:=0;
 			gvl.BLegSlip_trot_vel_desire:=0;
			gvl.BLegSlip_side_vel_desire:=0;
			gvl.BLegSlip_turn_rate_desire:=0;			
			IF trot_vel_desire=trot_vel AND side_vel_desire=side_vel AND turn_rate_desire=turn_rate THEN
				state:=ready;
				requir_stop:=FALSE;
				inSlip:=FALSE;
			END_IF
		END_IF
	END_IF
	IF state=ready THEN
		count_en_RD:=gait_cycle;
		tip_pos_en_RD:=tip_pos_ref;
		tip_vel_en_RD:=tip_vel_ref;	
	END_IF
END_IF
IF state=ready AND gait_cycle-count_en_RD=LREAL_TO_UDINT(2*gvl.sampleRate) THEN
	count_en_RD:=gait_cycle;
	tip_pos_en_RD:=tip_pos_ref;
	tip_vel_en_RD:=tip_vel_ref;	
END_IF

IF state<> state_last AND state=swing THEN
	Cmd2Tgt1Step(cmdVel:= trot_vel_desire, curVel:=trot_vel , step:= step[0], trgVel=>trot_vel );
	Cmd2Tgt1Step(cmdVel:= side_vel_desire, curVel:=side_vel , step:= step[1], trgVel=>side_vel );
	Cmd2Tgt1Step(cmdVel:= turn_rate_desire, curVel:=turn_rate , step:= step[2], trgVel=>turn_rate );
END_IF

state_last:=state; 
require_move_last:=require_move;
END_METHOD

METHOD PUBLIC TrjPlanning : BOOL
VAR_INPUT
END_VAR

VAR
	i: INT;
	FixTrj_tn:ARRAY[0..4] OF LREAL:=[0,0.25,0.5,0.75,1];
	InterplateValue:ARRAY[0..4] OF LREAL;
	InterplateTime:ARRAY[0..4] OF LREAL;
	start_vel:LREAL;
	end_vel:LREAL;
	j: INT;
	Rb_target1: Mat3;
	temp: vec3;
	Rb: Mat3;
	
	hip_pos_j : Vec3;
	leg_ref_pos_wrt_com_j : Vec3;
	tmp : Vec3;
	tip_pos, tip_vel : Vec3;
	jointTmpPosLast: ARRAY[0..2] OF LREAL;
END_VAR
gait_cycle := gait_cycle + 1;
IF state=swing THEN
	FOR i:=0 TO 4 DO
		SwingTrj_tn[i]:=FixTrj_tn[i]*period*(1-duty);
	END_FOR
	step_height_now :=step_height;
	FOR i:=0 TO 1 DO
		//trj planning in y direction (up/down)
		base_height:=normal_tip_pos_cart[1];
		start_height:=tip_pos_en_SW[i].data[1];
		InterplateValue[0]:=start_height;
		InterplateValue[1]:=(base_height * 0.05 + start_height * 0.95) + step_height_now * 0.6;
		InterplateValue[2]:=(base_height * 0.25 + start_height * 0.75) + step_height_now * 1.0;
		InterplateValue[3]:=(base_height * 0.65 + start_height * 0.35) + step_height_now * 0.6;
		InterplateValue[4]:=base_height;
		end_vel:=-0.01 / (period * duty);
		start_vel:=tip_vel_en_SW[i].data[1];
		fbCubicSpline(x:=SwingTrj_tn , y:=InterplateValue , dy0:=start_vel , dy4:=end_vel , 
			xt:=(gait_cycle-count_en_SW)*delta_t , yt=> tip_pos_ref[i].data[1], vt=> );
			
		 // trj planning in x direction (forward/backward)
		 base_x:=normal_tip_pos_cart[0];
		 trot_vel_now:=trot_vel-turn_rate*hip_pos[Mapping05[i],1];
		 step_length_now:= period * duty * trot_vel_now;
		 InterplateValue[0]:=tip_pos_en_SW[i].data[0];	
		 InterplateValue[1]:=base_x-0.48*step_length_now;;
		 InterplateValue[2]:=base_x;
		 InterplateValue[3]:=base_x+0.48*step_length_now;
		 InterplateValue[4]:=base_x+0.5*step_length_now;
		 end_vel:=-trot_vel_now;
		 start_vel:=tip_vel_en_SW[i].data[0];
		 fbCubicSpline(x:=SwingTrj_tn , y:=InterplateValue , dy0:=start_vel , dy4:=end_vel , 
			xt:=(gait_cycle-count_en_SW)*delta_t , yt=> tip_pos_ref[i].data[0], vt=> );
			
		 //trj planning in z direction (right/left)
		 base_z:=normal_tip_pos_cart[2];
		 //turn_vel_now:=turn_rate*(hip_pos[Mapping05[i],0]+normal_tip_pos_cart[1])+side_vel;
		 turn_vel_now:=turn_rate*(hip_pos[Mapping05[i],0]+normal_tip_pos_cart[0])+side_vel;
		 step_side_len_now := period * duty * turn_vel_now;
		 InterplateValue[0]:=tip_pos_en_SW[i].data[2];
		 InterplateValue[1]:=base_z+0.48* step_side_len_now;
		 InterplateValue[2]:=base_z;
		 InterplateValue[3]:=base_z-0.48* step_side_len_now;
		 InterplateValue[4]:=base_z-0.50* step_side_len_now;
		 end_vel:=turn_vel_now;
		 start_vel:=tip_vel_en_SW[i].data[2];
		 fbCubicSpline(x:=SwingTrj_tn , y:=InterplateValue , dy0:=start_vel , dy4:=end_vel , 
			xt:=(gait_cycle-count_en_SW)*delta_t , yt=> tip_pos_ref[i].data[2], vt=> );	
	END_FOR
ELSIF state=stance THEN 
	FOR i:=0 TO 4 DO
		StanceTrj_tn[i]:=FixTrj_tn[i]*period*duty;
	END_FOR
	FOR i:=0 TO 1 DO
		//trj planning in y direction (up/down)
		start_height:=tip_pos_en_ST[i].data[1];
		(*InterplateValue[0]:=start_height;
		InterplateValue[1]:=start_height-0.0045;
		InterplateValue[2]:=start_height-0.0085;
		InterplateValue[3]:=start_height-0.0125;
		InterplateValue[4]:=start_height-0.0160;*)
		InterplateValue[0]:=start_height;
		InterplateValue[1]:=start_height-0.0045*1;
		InterplateValue[2]:=start_height-0.0085*1;
		InterplateValue[3]:=start_height-0.0125*1;
		InterplateValue[4]:=start_height-0.0160*1;
		end_vel:=0;
		start_vel:=tip_vel_en_ST[i].data[1];
		fbCubicSpline(x:=StanceTrj_tn , y:=InterplateValue , dy0:=start_vel , dy4:=end_vel , 
			xt:=(gait_cycle-count_en_ST)*delta_t , yt=> tip_pos_ref[i].data[1], vt=> );	

		//trj planning in X direction (forward/backward)
		trot_vel_now:=trot_vel-	turn_rate*hip_pos[Mapping05[i],1];	
		step_length_now := period * duty * trot_vel_now;
		InterplateValue[0]:=tip_pos_en_ST[i].data[0];
		InterplateValue[1]:=tip_pos_en_ST[i].data[0]-0.28*step_length_now;
		InterplateValue[2]:=tip_pos_en_ST[i].data[0]-0.50*step_length_now;
		InterplateValue[3]:=tip_pos_en_ST[i].data[0]-0.72*step_length_now;
		InterplateValue[4]:=tip_pos_en_ST[i].data[0]-1.00*step_length_now;
		end_vel:= -trot_vel_now;
		start_vel:=tip_vel_en_ST[i].data[0];
		fbCubicSpline(x:=StanceTrj_tn , y:=InterplateValue , dy0:=start_vel , dy4:=end_vel , 
			xt:=(gait_cycle-count_en_ST)*delta_t , yt=> tip_pos_ref[i].data[0], vt=> );	
			
		// trj planning in z direction (right/left)
		//turn_vel_now:=turn_rate*(hip_pos[Mapping05[i],0]+normal_tip_pos_cart[1])+side_vel;
		turn_vel_now:=turn_rate*(hip_pos[Mapping05[i],0]+normal_tip_pos_cart[0])+side_vel;
		step_side_len_now := period * duty * turn_vel_now;
		InterplateValue[0]:=tip_pos_en_ST[i].data[2];
		InterplateValue[1]:=tip_pos_en_ST[i].data[2]+0.28*step_side_len_now;
		InterplateValue[2]:=tip_pos_en_ST[i].data[2]+0.50*step_side_len_now;
		InterplateValue[3]:=tip_pos_en_ST[i].data[2]+0.72*step_side_len_now;
		InterplateValue[4]:=tip_pos_en_ST[i].data[2]+1.00*step_side_len_now;
		end_vel:=turn_vel_now;
		start_vel:=tip_vel_en_ST[i].data[2];
		fbCubicSpline(x:=StanceTrj_tn , y:=InterplateValue , dy0:=start_vel , dy4:=end_vel , 
			xt:=(gait_cycle-count_en_ST)*delta_t , yt=> tip_pos_ref[i].data[2], vt=> );			
	END_FOR
ELSE
	FOR i:=0 TO 4 DO
		ReadyTrj_tn[i]:=FixTrj_tn[i]*2;//2s for ready gait
	END_FOR	
	FOR i:=0 TO 1 DO
		//trj planning in X direction (forward/backward)
		InterplateValue[0]:=tip_pos_en_RD[i].data[0];
		InterplateValue[1]:=tip_pos_en_RD[i].data[0];
		InterplateValue[2]:=tip_pos_en_RD[i].data[0];
		InterplateValue[3]:=tip_pos_en_RD[i].data[0];
		InterplateValue[4]:=tip_pos_en_RD[i].data[0];
		end_vel:=0;
		start_vel:=tip_vel_en_ST[i].data[0];
		fbCubicSpline(x:=ReadyTrj_tn , y:=InterplateValue , dy0:=start_vel , dy4:=end_vel , 
			xt:=(gait_cycle-count_en_RD)*delta_t , yt=> tip_pos_ref[i].data[0], vt=> );	

		//trj planning in y direction (right/left)
		InterplateValue[0]:=tip_pos_en_RD[i].data[1];
		InterplateValue[1]:=tip_pos_en_RD[i].data[1];
		InterplateValue[2]:=tip_pos_en_RD[i].data[1];
		InterplateValue[3]:=tip_pos_en_RD[i].data[1];
		InterplateValue[4]:=tip_pos_en_RD[i].data[1];
		end_vel:=0;
		start_vel:=tip_vel_en_ST[i].data[1];
		fbCubicSpline(x:=ReadyTrj_tn , y:=InterplateValue , dy0:=start_vel , dy4:=end_vel , 
			xt:=(gait_cycle-count_en_RD)*delta_t , yt=> tip_pos_ref[i].data[1], vt=> );	
		//trj planning in z direction (up/down)
		InterplateValue[0]:=tip_pos_en_RD[i].data[2];
		InterplateValue[1]:=tip_pos_en_RD[i].data[2];
		InterplateValue[2]:=tip_pos_en_RD[i].data[2];
		InterplateValue[3]:=tip_pos_en_RD[i].data[2];
		InterplateValue[4]:=tip_pos_en_RD[i].data[2];
		end_vel:=0;
		start_vel:=tip_vel_en_ST[i].data[2];
		fbCubicSpline(x:=ReadyTrj_tn , y:=InterplateValue , dy0:=start_vel , dy4:=end_vel , 
			xt:=(gait_cycle-count_en_RD)*delta_t , yt=> tip_pos_ref[i].data[2], vt=> );		
		END_FOR
END_IF
FOR i:=0 TO 1 DO
	FOR j:=0 TO 2 DO
		tip_vel_ref[i].data[j]:=(tip_pos_ref[i].data[j]-tip_pos_ref_last[i].data[j])/delta_t;
	END_FOR
END_FOR
tip_pos_ref_last:=tip_pos_ref;

body_ref_pos:=body_ref_pos_init;
body_ref_ang:=body_ref_ang_init;
leg_ref_pos:=leg_ref_pos_init;
FOR i:=0 TO 1 DO
	fbRotMat(yaw := body_ref_ang.data[2], pitch := body_ref_ang.data[1],roll := body_ref_ang.data[0], rm =>  Rb_target1 );
	temp.data[0]:=hip_pos[Mapping05[i],0];temp.data[1]:=hip_pos[Mapping05[i],1];temp.data[2]:=hip_pos[Mapping05[i],2];
	leg_ref_pos[Mapping05[i]]:= VecAdd( MatMulVec(Rb_target1, VecAdd(temp,MatMulVec(Rleg[Mapping05[i]],tip_pos_ref[i]))),body_ref_pos);
END_FOR

// transform TO leg local frame AND DO inverse kinematics

FOR j := 0 TO 5 DO
	fbRotMat(
    	yaw := body_ref_ang.data[2], 
		pitch := body_ref_ang.data[1], 
		roll := body_ref_ang.data[0], 
		rm => Rb);
	hip_pos_j := SetVec3(hip_pos[j, 0], hip_pos[j, 1], hip_pos[j, 2]);

	//leg_ref_pos_wrt_com = Rb' * (leg_ref_pos - body_ref_pos)
	leg_ref_pos_wrt_com_j := MatMulVec(
		                         MatTranspose(Rb),
								 VecAdd(
									 leg_ref_pos[j],
									 VecNeg(body_ref_pos)
                                 )
                             );
	// leg_ref_pos_wrt_hip = Rleg' * (leg_ref_pos_wrt_com_j - hip_pos)
	leg_ref_pos_next_wrt_hip[j] := MatMulVec(
		                               MatTranspose(Rleg[j]),
									   VecAdd(
										   leg_ref_pos_wrt_com_j,
										   VecNeg(hip_pos_j)
									   )
								   );
								   
	leg_ref_vel_next_wrt_hip[j] := VecMulNum(VecAdd(leg_ref_pos_next_wrt_hip[j], VecNeg(leg_ref_pos_wrt_hip[j])), DINT_TO_LREAL(gvl.sampleRate));
END_FOR


// mapping to actual joints
FOR j := 0 TO 5 DO
	tmp := leg_ref_pos_next_wrt_hip[leg_index_mapping[j]-1];
	tip_pos := SetVec3(tmp.data[0], tmp.data[1], tmp.data[2]);
	tmp := leg_ref_vel_next_wrt_hip[leg_index_mapping[j]-1];
	tip_vel := SetVec3(tmp.data[0], tmp.data[1], tmp.data[2]);
	FOR i:= 0 TO 2 DO
		jointTmpPosLast[i]:=jointPosLast[j,i];
	END_FOR		
	gvl.legCtrl[j].InversePosAndVel(
		tipPos := tip_pos.data, 
		tipVel := tip_vel.data, 
		refPosLast:=jointTmpPosLast,
		legIndex:=j,
		jntPos => joint_ref_pos[j].data, 
		jntVel => joint_ref_vel[j].data);
	
END_FOR

// link to physical outputs
FOR i := 0 TO 5 DO
	FOR j := 0 TO 2 DO
		jointPosTarget[i, j] := joint_ref_pos[i].data[j];
		jointPosLast[i,j]:=jointPosTarget[i, j] ;
		jointVelTarget[i, j] := joint_ref_vel[i].data[j];
		jointFceTarget[i, j] := 0;
	END_FOR
END_FOR

// store refs for next loop
leg_ref_pos_wrt_hip := leg_ref_pos_next_wrt_hip;
END_METHOD

END_FUNCTION_BLOCK

// ---- POUs/GaitPlanner/CurlingGaitFromSlip.TcPOU
FUNCTION_BLOCK CurlingGaitFromSlip
VAR_INPUT
END_VAR
VAR_OUTPUT
END_VAR
VAR
	tTotalAll     : LREAL := 5000;
	
	// robot geometrical parameters
	hip_pos : ARRAY[0..5, 0..2] OF LREAL := [-0.369,  -0.125, 0,
                                             0,  -0.28, 0,
                                             0.36, -0.125, 0,
                                             0.36, 0.125, 0,
											 0,0.28,0,
											 -0.369,0.125,0];

	leg_index_mapping : ARRAY[0..5] OF INT := [1, 2, 3, 4,5,6];
	Rleg : ARRAY[0..5] OF Mat3;
	
	gait_cycle : UDINT := 0;
	quit_flag : BOOL := FALSE;
	
	joint_ref_pos_init : ARRAY[0..5] OF Vec3;
	jointPosLast   : ARRAY[0..5, 0..2] OF LREAL; 
	
	body_ref_pos_init : Vec3;
	body_ref_ang_init : Vec3;
    leg_ref_pos_init : ARRAY[0..5] OF Vec3;
	leg_ref_pos_init_wrt_hip : ARRAY[0..5] OF Vec3;

	body_ref_pos : Vec3;
	body_ref_ang : Vec3;
	body_ref_angvel:vec3;
    leg_ref_pos : ARRAY[0..5] OF Vec3;
	leg_ref_pos_last : ARRAY[0..5] OF Vec3;
	leg_ref_pos_wrt_hip : ARRAY[0..5] OF Vec3;
	body_ref_pos_enter : Vec3;
	body_ref_ang_enter : Vec3;
    leg_ref_pos_enter : ARRAY[0..5] OF Vec3;
	leg_ref_pos_wrt_hip_enter : ARRAY[0..5] OF Vec3;
	
	body_ref_pos_next : Vec3;
	body_ref_ang_next : Vec3;
    leg_ref_pos_next : ARRAY[0..5] OF Vec3;
	leg_ref_pos_next_wrt_hip : ARRAY[0..5] OF Vec3;
	leg_ref_vel_next_wrt_hip : ARRAY[0..5] OF Vec3;
	
	// output test
	joint_ref_pos   : ARRAY[0..5] OF Vec3;
	joint_ref_vel   : ARRAY[0..5] OF Vec3;
	
	jointPosTarget  : ARRAY[0..5, 0..2] OF LREAL; 
	jointVelTarget  : ARRAY[0..5, 0..2] OF LREAL;  
	jointFceTarget  : ARRAY[0..5, 0..2] OF LREAL;  
	
	pvt, pvtDot : LREAL;
	
	fbRotmat : RotM;
	fbGetPivot  : GetPivot;
	delta_t:LREAL :=0.0025;//sample time
	
	isFinished : BOOL := FALSE;
	
	//target value from visual system
	adjust_angle_rad:LREAL:=0;//unit:rad
	adjust_angle_actual_rad:LREAL:=0;//unit:rad
	target_vel:LREAL:=0;//unit:m/s
	stone_rot_vel:LREAL:=0;//unit:rad/s
	
	//common variable
	sum_height : LREAL := 0;
	fbElipseInterpolation:ElipseInterpolation;
	fbHermitInterpolation:HermitInterpolation;
	Mapping14:ARRAY[0..1] OF INT:=[1,4];
	Mapping05:ARRAY[0..1] OF INT:=[0,5];
	Mapping23:ARRAY[0..1] OF INT:=[2,3];
	body_target_pos: Vec3;
	getPivot  : GetPivot;	
	tipForceDesire:ARRAY[0..5,0..2] OF LREAL;
	jntTrqDesire:ARRAY[0..5,0..2] OF LREAL;
	fceLoadTime:LREAL:=0.2;
	tipForceDesireZeros:ARRAY[0..5,0..2] OF LREAL:=[0,0,0,
													 0,0,0,
													 0,0,0,
													 0,0,0,
													 0,0,0,
													 0,0,0];
	tipForceTarget:		 ARRAY[0..5,0..2] OF LREAL:=[0,0,0,
													 0,0,0,
													 0,0,0,
													 0,0,0,
													 0,0,0,
													 0,0,0];	
	
	//state machine 
	state:UINT;
	Ready:UINT:=1;//init state
	MlegRollA:UINT:=3;
	BodyPosAdjust:UINT:=6;
	BLegPosAdjust:UINT:=7;
	SearchPedal:UINT:=8;
	ArmControl:UINT:=9;
	OrientAdjust:UINT:=10;
	MlegRollB:UINT:=11;
	StoneRot:UINT:=12;
	LiftMleg:UINT:=13;
	SpeedUp:UINT:=14;
	Slide:UINT:=15;
	PushReleaseBall:UINT:=16;
	SpeedDown:UINT:=17;
	BLegRecovery:UINT:=18;
	MlegRollC:UINT:=19;
	AddHeight:UINT:=20;
	FlegRotB:UINT:=21;
	Recovery:UINT:=22;
	CurlingFinished:UINT:=23;
	
	//contol button
	RequireMlegRollA:BOOL:=FALSE;
	RequireBodyPosAdjust:BOOL:=FALSE;
	RequireBLegPosAdjust:BOOL:=FALSE;
	RequireSearchPedal:BOOL:=FALSE;
	RequireArmControl:BOOL:=FALSE;
	RequireOrientAdjust:BOOL:=FALSE;
	RequireMlegRollB:BOOL:=FALSE;	
	RequireStoneRot:BOOL:=FALSE;		
	RequireLiftMleg:BOOL:=FALSE;
	RequireSpeedUp:BOOL:=FALSE;
	RequireSlide:BOOL:=FALSE;
	RequirePushReleaseBall:BOOL:=FALSE;
	RequireSpeedDown:BOOL:=FALSE;
	RequireBLegRecovery:BOOL:=FALSE;
	RequireMlegRollC:BOOL:=FALSE;
	RequireAddHeight:BOOL:=FALSE;
	RequireFlegRotB:BOOL:=FALSE;
	RequireRecovery:BOOL:=FALSE;
	
	RequireRepeateBodyPosAdjust:BOOL:=FALSE;
	RequireRepeateBLegPosAdjust:BOOL:=FALSE;
	RequireRepeateSearchPedal:BOOL:=FALSE;
	RequireRepeateArmControl:BOOL:=FALSE;
	RequireRepeateOrientAdjust:BOOL:=FALSE;
	RequireRepeateStoneRot:BOOL:=FALSE;
	
	IsReady:BOOL:=FALSE;
	IsMlegRollA:BOOL:=FALSE;
	IsBodyPosAdjust:BOOL:=FALSE;
	IsBLegPosAdjust:BOOL:=FALSE;
	IsSearchPedal:BOOL:=FALSE;
	IsArmControl:BOOL:=FALSE;
	IsOrientAdjust:BOOL:=FALSE;
	IsMlegRollB:BOOL:=FALSE;	
	IsStoneRot:BOOL:=FALSE;		
	IsLiftMleg:BOOL:=FALSE;
	IsSpeedUp:BOOL:=FALSE;
	IsSlide:BOOL:=FALSE;
	IsPushReleaseBall:BOOL:=FALSE;
	IsSpeedDown:BOOL:=FALSE;
	IsBLegRecovery:BOOL:=FALSE;
	IsMlegRollC:BOOL:=FALSE;
	IsAddHeight:BOOL:=FALSE;
	IsFlegRotB:BOOL:=FALSE;
	IsRecovery:BOOL:=FALSE;
	IsCurlingFinished:BOOL:=FALSE;

	ReadyFinished:bool:=false;
	MlegRollAFinished:BOOL:=FALSE;
	BodyPosAdjustFinished:BOOL:=FALSE;
	BLegPosAdjustFinished:BOOL:=FALSE;	
	SearchPedalFinished:BOOL:=FALSE;
	ArmControlFinished:BOOL:=FALSE;
	OrientAdjustFinished:BOOL:=FALSE;
	MlegRollBFinished:BOOL:=FALSE;
	StoneRotFinished:BOOL:=FALSE;
	LiftMlegFinished:BOOL:=FALSE;
	SpeedUpFinished:BOOL:=FALSE;
	SlideFinished:BOOL:=FALSE;
	PushReleaseBallFinished:BOOL:=FALSE;
	SpeedDownFinished:BOOL:=FALSE;
	BLegRecoveryFinished:BOOL:=FALSE;
	MlegRollCFinished:BOOL:=FALSE;
	AddHeightFinished:BOOL:=FALSE;
	FlegRotBFinished:BOOL:=FALSE;
	RecoveryFinished:BOOL:=FALSE;
	CurlingGaitFinished: BOOL:=FALSE;
	
	EnterMlegRollACount:UDINT;
	EnterBodyPosAdjustCount:UDINT;
	EnterBLegPosAdjustCount:UDINT;
	EnterSearchPedalCount:UDINT;
	EnterArmControlCount:UDINT;
	EnterOrientAdjustCount:UDINT;
	EnterMlegRollBCount:UDINT;
	EnterStoneRotCount:UDINT;
	EnterLiftMlegCount:UDINT;
	EnterSpeedUpCount:UDINT;
	EnterSlideCount:UDINT;
	EnterPushReleaseBallCount:UDINT;
	EnterSpeedDownCount:UDINT;
	EnterBLegRecoveryCount:UDINT;
	EnterMlegRollCCount:UDINT;
	EnterAddHeightCount:UDINT;
	EnterFlegRotBCount:UDINT;
	EnterRecoveryCount:UDINT;
	
	//MlegRollA
	MlegRollA_MJntStart:ARRAY[0..1] OF vec3;
	MlegRollA_MPosWrtHip:ARRAY[0..1] OF vec3;
	MlegRollA_MJntRef:ARRAY[0..1] OF vec3;
	MlegRollATime:LREAL:=3;
	MlegRollA_MJntTarget:ARRAY[0..1,0..2] OF LREAL;
	
	//BodyPosAdjust
	BPA_x:LREAL:=0;
	BPA_y:LREAL:=0;
	BPA_AngRad:LREAL:=0;
	BPA_HeightAdd:LREAL:=0.05;
	BPA_RotCenter1:vec3;
	BPA_BodyPosStart:vec3;
	BPA_BodyAngStart:vec3;
	BPA_BodyPoseEnd:vec3;
	BPA_BodyAngEnd:vec3;
	BPA_LiftGroundTime:LREAL:=1;
	BPA_AdjustTime:LREAL:=1;
	BPA_AdjustExtractTime:LREAL:=0.5;
	BPA_AdjustExtendTime:LREAL:=0.5;
	BPA_FJntRef:ARRAY[0..1] OF vec3;
	BPA_FPosWrtHip:ARRAY[0..1] OF vec3;
	BPA_MJntStart:ARRAY[0..1] OF vec3;
	BPA_MJntRef:ARRAY[0..1] OF vec3;
	BPA_MPosWrtHip:ARRAY[0..1] OF vec3;
	BPA_MJntExtend:ARRAY[0..1,0..2] OF LREAL;
	BPA_MJntExtract:ARRAY[0..1,0..2] OF LREAL;	
	BPA_BJntStart:ARRAY[0..1] OF vec3;
	BPA_BJntRef:ARRAY[0..1] OF vec3;
	BPA_BPosWrtHip:ARRAY[0..1] OF vec3;
	BPA_BJntExtend:ARRAY[0..1,0..2] OF LREAL;
	BPA_BJntExtract:ARRAY[0..1,0..2] OF LREAL;	
	BPA_legPosEnterExtract:ARRAY[0..5] OF vec3;
	
	//BLegPosAdjust
	BLPA_adjust_distance:ARRAY[0..1,0..2] OF LREAL:=[0,0,0,0,0,0];
	BLPA_tgtLegPos:ARRAY[0..5] OF vec3;
	BLPA_time:LREAL:=1;
	BLPA_height:LREAL:=0.05;
	leg_ref_pos_enter_next:ARRAY[0..5] OF vec3;
	
	//search pedal
	SP_RBLegSearching:BOOL:=FALSE;
	SP_LBLegSearching:BOOL:=FALSE;
	SP_EnterSubSearchCount:ARRAY[0..1] OF UDINT;
	SP_EnterSubSearchDecreaseCount:ARRAY[0..1] OF UDINT;
	SP_BLegSearchFinished:ARRAY [0..1] OF BOOL:=[FALSE,FALSE];
	
	SP_PedalSearched:ARRAY [0..1] OF BOOL:=[FALSE,FALSE];
	SP_BJntStart:ARRAY[0..1] OF vec3;
	SP_BPosStartWrtHip:ARRAY[0..1] OF vec3;
	SP_BPosRefWrtHip:ARRAY[0..1] OF vec3;
	SP_BPosLockWrtHip:ARRAY[0..1] OF vec3;
	SP_LiftLegTime:LREAL:=0.5;
	SP_LiftDistance:LREAL:=0.03;
	SP_SearchTime:LREAL:=3;
	SP_SearchDistance:LREAL:=0.05;
	
	//ArmControl
	AC_time:LREAL:=5;
	AC_AngleDeg:LREAL:=-15;
	AC_AngleRad:LREAL:=-15*pi/180;
	AC_Velocity:LREAL;
	AC_extend:BOOL:=FALSE;
	AC_retract:BOOL:=FALSE;
	AC_wait:BOOL:=FALSE;
	AC_EnterExtendCount:UDINT;
	AC_EnterRetractCount:UDINT;

	//OrientAdjust
	OA_HeighAdd:LREAL:=0.05;
	OA_RotCenter1:vec3;
	OA_BodyPosStart:vec3;
	OA_BodyAngStart:vec3;
	OA_BodyPoseEnd:vec3;
	OA_BodyAngEnd:vec3;
	OA_LiftGroundTime:LREAL:=1;
	OA_AdjustTime:LREAL:=1;
	OA_AdjustExtractTime:LREAL:=0.5;
	OA_AdjustExtendTime:LREAL:=0.5;
	OA_FJntRef:ARRAY[0..1] OF vec3;
	OA_FPosWrtHip:ARRAY[0..1] OF vec3;
	OA_MJntStart:ARRAY[0..1] OF vec3;
	OA_MJntRef:ARRAY[0..1] OF vec3;
	OA_MPosWrtHip:ARRAY[0..1] OF vec3;
	OA_legPosEnterExtract:ARRAY[0..5] OF vec3;
	OA_MJntExtend:ARRAY[0..1,0..2] OF LREAL;
	OA_MJntExtract:ARRAY[0..1,0..2] OF LREAL;
	
	//MlegRollB
	MlegRollB_MJntStart:ARRAY[0..1] OF vec3;
	MlegRollB_MPosWrtHip:ARRAY[0..1] OF vec3;
	MlegRollB_MJntRef:ARRAY[0..1] OF vec3;
	MlegRollBTime:LREAL:=3;
	MlegRollB_MJntTarget:ARRAY[0..1,0..2] OF LREAL;
	
	//StoneRot
	StoneRot_FJntStart:ARRAY[0..1] OF vec3;
	StoneRot_FPosWrtHip:ARRAY[0..1] OF vec3;
	StoneRot_FJntRef:ARRAY[0..1] OF vec3;
	StoneGripTime:LREAL:=1;
	SetColide:BOOL:=FALSE;
	StoneRotSubState:ARRAY [0..1] OF BOOL:=[FALSE,FALSE];
	StoneRotTime:LREAL:=2;
	
	//LiftMleg
	LiftMleg_MJntStart:ARRAY[0..1] OF vec3;
	LiftMleg_MJntRef:ARRAY[0..1] OF vec3;
	LiftMleg_MPosWrtHip:ARRAY[0..1] OF vec3;
	LiftMlegTime:LREAL:=0.5;
	
	//SpeedUp
	SpeedUpSubState:UINT:=0;
	SpeedUpAS:UINT:=1;//acceleration
	SpeedUpCS:UINT:=2;//constant velocity
	SpeedUpDS:UINT:=3;//deceleration velocity
	SpeedUpSS:UINT:=4;//stop
	 
	//Distance_x_AS:LREAL:=0.3;// acceleration distance in x direction
	Distance_x_AS:LREAL:=0.3;// acceleration distance in x direction
	Distance_x_DS:LREAL:=0.05;// deceleration distance in x direction
	Distance_y_DS:LREAL:=0.1;// deceleration distance in y direction 0.05
	Distance_x_total:LREAL:=0.6;//total extend length
	Time_AS:LREAL:=0.5;//acceleration time
	Time_CS:LREAL:=0.05;//constant time
	Time_DS:LREAL:=0.2;//deceleration time
	CurrentBLegMaxDistance:lreal;
	 
	EnterSpeedUpASCount:UDINT;
	EnterSpeedUpCSCount:UDINT;
	EnterSpeedUpDSCount:UDINT;
	EnterSpeedUpSPCount:UDINT;
	
	SpeedUp_MJntRef:ARRAY[0..1] OF vec3;
	SpeedUp_MPosWrtHip:ARRAY[0..1] OF vec3;
	SpeedUp_FJntRef:ARRAY[0..1] OF vec3;
	SpeedUp_FPosWrtHip:ARRAY[0..1] OF vec3;
	SpeedUp_BJntStart:ARRAY[0..1] OF vec3;
	SpeedUp_BPosWrtHipStart:ARRAY[0..1] OF vec3;
	
	body_ref_pos_wrt_body:vec3;
	
	//Slide
	slideTime:lreal:=0.3;
	
	//PushReleaseBall
	PushReleaseBall_FJntStart:ARRAY[0..1] OF vec3;
	PushReleaseBall_FPosStartWrtHip:ARRAY[0..1] OF vec3;
	PushReleaseBall_FJntRef:ARRAY[0..1] OF vec3;
	PushReleaseBall_FPosWrtHip:ARRAY[0..1] OF vec3;
	PRDistance_x_total:LREAL:=0.3;
	PushTime:LREAL:=0.2;
	PushDistance:LREAL:=0.2;
	PRConstVelDistance:LREAL:=0.05;
	PRConstVelTime:LREAL:=0.05;
	DecVelTime:LREAL:=0.1;
	DecVelDistance:LREAL:=0.05;
	PushVelocity:LREAL:=0.5;
	ReleaseTime:LREAL:=0.25;
	EnterPushFinishCount:UDINT;
	PushFinishDurationTime:LREAL:=2;
	
	//SpeedDown
	SpeedDownTime:LREAL:=0.5;
	SpeedDown_MJntStart:ARRAY[0..1] OF vec3;
	SpeedDown_MJntRef:ARRAY[0..1] OF vec3;
	SpeedDown_MPosWrtHip:ARRAY[0..1] OF vec3;	
	SpeedDown_MJntTarget:ARRAY[0..1,0..2] OF LREAL;
	
	//BLegRecovery
	BLRRetractTime:LREAL:=1.5;
	BLRExtendTime:LREAL:=1.5;
	BLR_FJntStart:ARRAY[0..1] OF vec3;
	BLR_FJntRef:ARRAY[0..1] OF vec3;
	BLR_FPosWrtHip:ARRAY[0..1] OF vec3;
	BLR_FJntExtractTarget:ARRAY[0..1,0..2] OF LREAL;
	BLR_FJntExtendTarget:ARRAY[0..1,0..2] OF LREAL;
	
	//MlegRollC
	MlegRollC_MJntStart:ARRAY[0..1] OF vec3;
	MlegRollC_MPosWrtHip:ARRAY[0..1] OF vec3;
	MlegRollC_MJntRef:ARRAY[0..1] OF vec3;
	MlegRollCTime:LREAL:=3;
	MlegRollC_MJntTarget:ARRAY[0..1,0..2] OF LREAL;
	
	//AddHeight
	AddHeightTime:LREAL:=1;
	AddHeight_FJntStart:ARRAY[0..1] OF vec3;
	AddHeight_FPosWrtHip:ARRAY[0..1] OF vec3;
	
	//FlegRotB
	FlegRotBTime:LREAL:=2;
	FlegRotB_FJntStart:ARRAY[0..1] OF vec3;
	FlegRotB_FJntRef:ARRAY[0..1] OF vec3;
	FlegRotB_FPosWrtHip:ARRAY[0..1] OF vec3;	
	
	//recovery
	RcJointPosStart   : ARRAY[0..5, 0..2] OF LREAL; 
	jntAngRetract:ARRAY[0..5,0..2] OF LREAL	;
	jntAngExtend:ARRAY[0..5,0..2] OF LREAL;	
	tRetract   : LREAL := 3;
	tWait      : LREAL := 1;
	tExtend    : LREAL := 3;	
	pivot, pivotDot : LREAL;
	RcJointPosRef:ARRAY[0..5,0..2] OF LREAL;	
	Rc_PosWrtHip:ARRAY[0..5] OF vec3;
	FlegRotB_FJntState3:ARRAY[0..1,0..2] OF LREAL;
	
END_VAR

METHOD PUBLIC DoPlanning : BOOL
VAR_INPUT
	count : UDINT;
END_VAR
VAR
	i, j  : INT;
END_VAR
IF count = 0 THEN
	isFinished := FALSE;
	Initialize();
END_IF

IF RequireRepeateStoneRot=TRUE AND StoneRotFinished=TRUE AND state=StoneRot THEN
	state:=MlegRollB;
    MlegRollBFinished:=TRUE;
    RequireStoneRot:=TRUE;
	RequireRepeateStoneRot:=FALSE;
END_IF

IF RequireRepeateBodyPosAdjust=TRUE AND state=BodyPosAdjust AND BodyPosAdjustFinished=TRUE THEN
	state:=MlegRollA;
    MlegRollAFinished:=TRUE; 
	RequireBodyPosAdjust:=TRUE;
	RequireRepeateBodyPosAdjust:=FALSE;
END_IF
IF RequireRepeateBLegPosAdjust=TRUE AND state=BLegPosAdjust AND BLegPosAdjustFinished=TRUE THEN
	state:=BodyPosAdjust;
    BodyPosAdjustFinished:=TRUE; 
	RequireBLegPosAdjust:=TRUE;
	RequireRepeateBLegPosAdjust:=FALSE;
END_IF

IF RequireRepeateSearchPedal=TRUE AND state=SearchPedal AND SearchPedalFinished=TRUE THEN
	state:=BLegPosAdjust;
    BLegPosAdjustFinished:=TRUE; 
	RequireSearchPedal:=TRUE;
	RequireRepeateSearchPedal:=FALSE;
END_IF

IF RequireRepeateArmControl=TRUE AND state=ArmControl AND ArmControlFinished=TRUE THEN
	state:=SearchPedal;
    SearchPedalFinished:=TRUE; 
	RequireArmControl:=TRUE;
	RequireRepeateArmControl:=FALSE;
END_IF

IF RequireRepeateOrientAdjust=TRUE AND state=OrientAdjust AND OrientAdjustFinished=TRUE THEN
	state:=BLegPosAdjust;
    BLegPosAdjustFinished:=TRUE; 
	RequireOrientAdjust:=TRUE;
	RequireRepeateOrientAdjust:=FALSE;
END_IF

StateMachine();
TrjPlanning();

IF quit_flag THEN
	isFinished := TRUE;
	quit_flag := FALSE;
	
	RequireMlegRollA:=FALSE;
	RequireBodyPosAdjust:=FALSE;
	RequireBLegPosAdjust:=FALSE;
	RequireSearchPedal:=FALSE;
	RequireArmControl:=FALSE;
	RequireOrientAdjust:=FALSE;
	RequireMlegRollB:=FALSE;	
	RequireStoneRot:=FALSE;		
	RequireLiftMleg:=FALSE;
	RequireSpeedUp:=FALSE;
	RequireSlide:=FALSE;
	RequirePushReleaseBall:=FALSE;
	RequireSpeedDown:=FALSE;
	RequireBLegRecovery:=FALSE;
	RequireMlegRollC:=FALSE;
	RequireAddHeight:=FALSE;
	RequireFlegRotB:=FALSE;

	MlegRollAFinished:=FALSE;
	BodyPosAdjustFinished:=FALSE;
	BLegPosAdjustFinished:=FALSE;
	SearchPedalFinished:=FALSE;
	ArmControlFinished:=FALSE;
	OrientAdjustFinished:=FALSE;
	MlegRollBFinished:=FALSE;
	StoneRotFinished:=FALSE;
	LiftMlegFinished:=FALSE;
	SpeedUpFinished:=FALSE;
	SlideFinished:=FALSE;
	PushReleaseBallFinished:=FALSE;
	SpeedDownFinished:=FALSE;
	MlegRollCFinished:=FALSE;
	BLegRecoveryFinished:=FALSE;
	AddHeightFinished:=FALSE;
	FlegRotBFinished:=FALSE;
	RecoveryFinished:=FALSE;
	CurlingGaitFinished:=FALSE;
	
	RequireRepeateBodyPosAdjust:=FALSE;
	RequireRepeateSearchPedal:=FALSE;
	RequireRepeateBLegPosAdjust:=FALSE;
	RequireRepeateOrientAdjust:=FALSE;
	RequireRepeateStoneRot:=FALSE;
END_IF
END_METHOD

METHOD PUBLIC Initialize : BOOL
VAR_INPUT
END_VAR
VAR
	i, j : INT;
	
	leg_pos    : ARRAY[0..2] OF LREAL;
	
	Rb : Mat3;
	hip_pos_j  : Vec3;
	leg_pos_wrt_com : Vec3;
	
END_VAR
Rleg[0]:=SetMat3(1,0,0,0,0,-1,0,1,0);
Rleg[1]:=SetMat3(-1,0,0,0,0,1,0,1,0,);
Rleg[2]:=SetMat3(-1,0,0,0,0,1,0,1,0);
Rleg[3]:=SetMat3(-1,0,0,0,0,1,0,1,0);
Rleg[4]:=SetMat3( -1,0,0,0,0,1,0,1,0);
Rleg[5]:=SetMat3(1,0,0,0,0,-1,0,1,0);

state:=Ready;
ReadyFinished:=true;
quit_flag  := FALSE;
gait_cycle := 0;

// control button for each state, need be commented out at actual environment
RequireMlegRollA:=FALSE;
RequireBodyPosAdjust:=FALSE;
RequireBLegPosAdjust:=FALSE;
RequireSearchPedal:=FALSE;
RequireArmControl:=FALSE;
RequireOrientAdjust:=FALSE;
RequireMlegRollB:=FALSE;	
RequireStoneRot:=FALSE;		
RequireLiftMleg:=FALSE;
RequireSpeedUp:=FALSE;
RequireSlide:=FALSE;
RequirePushReleaseBall:=FALSE;
RequireSpeedDown:=FALSE;
RequireBLegRecovery:=FALSE;
RequireMlegRollC:=FALSE;
RequireAddHeight:=FALSE;
RequireFlegRotB:=FALSE;

MlegRollAFinished:=FALSE;
BodyPosAdjustFinished:=FALSE;
BLegPosAdjustFinished:=FALSE;
SearchPedalFinished:=FALSE;
ArmControlFinished:=FALSE;
OrientAdjustFinished:=FALSE;
MlegRollBFinished:=FALSE;
StoneRotFinished:=FALSE;
LiftMlegFinished:=FALSE;
SpeedUpFinished:=FALSE;
SlideFinished:=FALSE;
PushReleaseBallFinished:=FALSE;
SpeedDownFinished:=FALSE;
BLegRecoveryFinished:=FALSE;
MlegRollCFinished:=FALSE;
AddHeightFinished:=FALSE;
FlegRotBFinished:=FALSE;
CurlingGaitFinished:=FALSE;

RequireRepeateBodyPosAdjust:=FALSE;
RequireRepeateBLegPosAdjust:=FALSE;
RequireRepeateSearchPedal:=FALSE;
RequireRepeateArmControl:=FALSE;
RequireRepeateOrientAdjust:=FALSE;
RequireRepeateStoneRot:=FALSE;

// bodyRot
delta_t:=1.0/gvl.SampleRate;//sample time
SetTargetValue(GVL.adjust_angle_degree,GVL.target_vel,GVL.stone_rot_vel);
IsReady:=true;

FOR i := 0 TO 5 DO
	FOR j := 0 TO 2 DO
		IF ABS(gvl.jntLastRefPos[i, j] - gvl.jntActualPos[i, j]) < gvl.curling_threshold_value THEN
			joint_ref_pos_init[i].data[j] := gvl.jntLastRefPos[i, j];
		ELSE
			joint_ref_pos_init[i].data[j] := gvl.jntActualPos[i, j];
		END_IF
		jointPosLast[i,j]:=joint_ref_pos_init[i].data[j];
	END_FOR
END_FOR

(*FOR i := 0 TO 5 DO
	FOR j := 0 TO 2 DO
		joint_ref_pos_init[i].data[j] := gvl.jntActualPos[i, j];
		jointPosLast[i,j]:=joint_ref_pos_init[i].data[j];
	END_FOR
END_FOR*)

sum_height := 0;
FOR j := 0 TO 5 DO
	// FK
	gvl.legCtrl[j].ForwardKinetics(motorAngles := joint_ref_pos_init[j].data, legIndex:=j, tipPosition => leg_pos);
	leg_ref_pos_init_wrt_hip[j] := SetVec3(leg_pos[0], leg_pos[1], leg_pos[2]);
	sum_height := sum_height - leg_ref_pos_init_wrt_hip[j].data[1];
END_FOR
body_ref_pos_init := SetVec3(0, 0, sum_height/6.0);
body_ref_ang_init := SetVec3(0, 0, 0);                            

FOR j := 0 TO 5 DO
	fbRotMat(yaw := body_ref_ang_init.data[2],
             pitch := body_ref_ang_init.data[1],
             roll := body_ref_ang_init.data[0],
             rm => Rb );
	hip_pos_j := SetVec3(hip_pos[j, 0], hip_pos[j, 1], hip_pos[j, 2]);
	leg_pos_wrt_com := VecAdd(MatMulVec(Rleg[j], leg_ref_pos_init_wrt_hip[j]), hip_pos_j);
    leg_ref_pos_init[j] := VecAdd(body_ref_pos_init, MatMulVec(Rb, leg_pos_wrt_com));
END_FOR

body_ref_pos := body_ref_pos_init;
body_ref_ang := body_ref_ang_init;
leg_ref_pos := leg_ref_pos_init;
leg_ref_pos_wrt_hip := leg_ref_pos_init_wrt_hip;
leg_ref_pos_last:=leg_ref_pos;

FOR i := 0 TO 5 DO
	FOR j := 0 TO 2 DO
		jointPosTarget[i, j] := joint_ref_pos_init[i].data[j];
		jointVelTarget[i, j] := 0;
		jointFceTarget[i, j] := 0;
	END_FOR
END_FOR
END_METHOD

METHOD PUBLIC isPedal : BOOL
VAR_INPUT
		legIndex:INT;
END_VAR
IF ABS(gvl.tipActualFce[legIndex,0])>40 THEN //10 need be calibrated
	isPedal:=TRUE;
ELSE
	isPedal:=FALSE;
END_IF
END_METHOD

METHOD PUBLIC isStone : BOOL
VAR_INPUT
	legIndex:INT;
END_VAR
IF ABS(gvl.tipActualFce[legIndex,2])>50 THEN //10 need be calibrated
	isStone:=TRUE;
ELSE
	isStone:=FALSE;
END_IF
END_METHOD

METHOD PUBLIC SetTargetValue : BOOL
VAR_INPUT
	in_adjust_angle_degree:LREAL:=0;//unit:degree
	in_target_vel:LREAL:=0;//unit:m/s
	in_stone_rot_vel:LREAL:=0;//unit:rpm
END_VAR
adjust_angle_rad:=in_adjust_angle_degree*pi/180;
target_vel:=in_target_vel;
stone_rot_vel:=in_stone_rot_vel/60*2*pi;
END_METHOD

METHOD PUBLIC StateMachine : BOOL
VAR_INPUT
END_VAR

VAR
	i: INT;
	j: INT;
	RotRadius: LREAL;
END_VAR
IF state=ready AND RequireMlegRollA=TRUE THEN
	state:=MlegRollA;
	IsReady:=FALSE;
	IsMlegRollA:=TRUE;
	RequireMlegRollA:=FALSE;
	body_ref_pos_enter := body_ref_pos;
	body_ref_ang_enter := body_ref_ang;
	leg_ref_pos_enter := leg_ref_pos;
	EnterMlegRollACount:=gait_cycle;
	MlegRollAFinished:=FALSE;
	FOR i:=0 TO 1 DO
		FOR j:=0 TO 2 DO
			MlegRollA_MJntStart[i].data[j]:=jointPosLast[Mapping14[i],j];
		END_FOR
	END_FOR
ELSIF state=MlegRollA AND MlegRollAFinished=TRUE AND RequireBodyPosAdjust=TRUE THEN
	state:=BodyPosAdjust;
	IsMlegRollA:=FALSE;
	IsBodyPosAdjust:=TRUE;
	requireBodyPosAdjust:=FALSE;
	body_ref_pos_enter := body_ref_pos;
	body_ref_ang_enter := body_ref_ang;
	leg_ref_pos_enter := leg_ref_pos;
	EnterBodyPosAdjustCount:=gait_cycle;
	BodyPosAdjustFinished:=FALSE;		
	FOR i:=0 TO 1 DO
		FOR j:=0 TO 2 DO
			BPA_FJntRef[i].data[j]:=jointPosLast[Mapping23[i],j];
			BPA_MJntExtend[i,j]:=jointPosLast[Mapping14[i],j];
			BPA_BJntExtend[i,j]:=jointPosLast[Mapping05[i],j];
		END_FOR
		BPA_MJntExtract[i,0]:=BPA_MJntExtend[i,0];
		BPA_MJntExtract[i,1]:=BPA_MJntExtend[i,1]-10*pi/180.0;
		BPA_MJntExtract[i,2]:=BPA_MJntExtend[i,2]+10*pi/180.0;
		BPA_BJntExtract[i,0]:=BPA_BJntExtend[i,0];
		BPA_BJntExtract[i,1]:=BPA_BJntExtend[i,1]-10*pi/180.0;
		BPA_BJntExtract[i,2]:=BPA_BJntExtend[i,2]+10*pi/180.0;
	END_FOR	
	FOR i:=0 TO 2 DO
		BPA_RotCenter1.data[i]:=0.5*(leg_ref_pos_enter[0].data[i]+leg_ref_pos_enter[5].data[i]);
	END_FOR	
	BPA_BodyPosStart:=body_ref_pos_enter;
	BPA_BodyAngStart:=body_ref_ang_enter;	
	RotRadius:=SQRT((BPA_BodyPosStart.data[0]-BPA_RotCenter1.data[0])*(BPA_BodyPosStart.data[0]-BPA_RotCenter1.data[0])+
				(BPA_BodyPosStart.data[1]-BPA_RotCenter1.data[1])*(BPA_BodyPosStart.data[1]-BPA_RotCenter1.data[1]));	
	BPA_AngRad:=GVL.BPA_adjust_angle_degree*pi/180;
	BPA_x:=gvl.BPA_adjust_x;
	BPA_y:=gvl.BPA_adjust_y;
	BPA_BodyPoseEnd.data[0]:=BPA_RotCenter1.data[0]+RotRadius*COS(BPA_AngRad+BPA_BodyAngStart.data[2])+BPA_x;
	BPA_BodyPoseEnd.data[1]:=BPA_RotCenter1.data[1]+RotRadius*SIN(BPA_AngRad+BPA_BodyAngStart.data[2])+BPA_y;
	BPA_BodyPoseEnd.data[2]:=body_ref_pos_enter.data[2];
	BPA_BodyAngEnd:=BPA_BodyAngStart;
	BPA_BodyAngEnd.data[2]:=BPA_BodyAngStart.data[2]+BPA_AngRad;	
ELSIF state=BodyPosAdjust AND BodyPosAdjustFinished=TRUE AND RequireBLegPosAdjust=TRUE THEN
	state:=BLegPosAdjust;
	IsBodyPosAdjust:=FALSE;
	IsBLegPosAdjust:=TRUE;
	requireBLegPosAdjust:=FALSE;
	body_ref_pos_enter := body_ref_pos;
	body_ref_ang_enter := body_ref_ang;
	leg_ref_pos_enter := leg_ref_pos;
	EnterBLegPosAdjustCount:=gait_cycle;
	BLegPosAdjustFinished:=FALSE;	
	
